LIN {X 0,Y 490.611,Z 701.735,A -85,B 0,C 180,E1 -6449.611,E2 -6449.611} C_VEL
LIN {X 0,Y 490.925,Z 689.002,A -85,B 0,C 180,E1 -6450.162,E2 -6450.162} C_VEL
LIN {X 0,Y 491.127,Z 676.229,A -85,B 0,C 180,E1 -6450.536,E2 -6450.536} C_VEL
LIN {X 0,Y 491.315,Z 653.215,A -85,B 0,C 180,E1 -6450.913,E2 -6450.913} C_VEL
LIN {X 0,Y 491.695,Z 579.169,A -85,B 0,C 180,E1 -6452.03,E2 -6452.03} C_VEL
LIN {X 0,Y 489.54,Z 572.056,A -85,B 0,C 180,E1 -6452.216,E2 -6452.216} C_VEL
LIN {X 0,Y 488.77,Z 569.605,A -85,B 0,C 180,E1 -6452.285,E2 -6452.285} C_VEL
LIN {X 0,Y 488.731,Z 569.605,A -85,B 0,C 180,E1 -6455.353,E2 -6455.353} C_VEL
LIN {X 0,Y 488.692,Z 569.612,A -85,B 0,C 180,E1 -6458.043,E2 -6458.043} C_VEL
LIN {X 0,Y 488.737,Z 569.609,A -85,B 0,C 180,E1 -6460.686,E2 -6460.686} C_VEL
LIN {X 0,Y 488.723,Z 569.605,A -85,B 0,C 180,E1 -6463.285,E2 -6463.285} C_VEL
LIN {X 0,Y 488.731,Z 569.605,A -85,B 0,C 180,E1 -6465.85,E2 -6465.85} C_VEL
LIN {X 0,Y 488.823,Z 569.598,A -85,B 0,C 180,E1 -6468.388,E2 -6468.388} C_VEL
LIN {X 0,Y 488.809,Z 569.594,A -85,B 0,C 180,E1 -6471.733,E2 -6471.733} C_VEL
LIN {X 0,Y 488.861,Z 569.591,A -85,B 0,C 180,E1 -6474.224,E2 -6474.224} C_VEL
LIN {X 0,Y 488.952,Z 569.573,A -85,B 0,C 180,E1 -6477.529,E2 -6477.529} C_VEL
LIN {X 0,Y 488.959,Z 569.576,A -85,B 0,C 180,E1 -6480,E2 -6480} C_VEL
LIN {X 0,Y 488.952,Z 569.583,A -85,B 0,C 180,E1 -6482.471,E2 -6482.471} C_VEL
LIN {X 0,Y 488.863,Z 569.586,A -85,B 0,C 180,E1 -6485.776,E2 -6485.776} C_VEL
LIN {X 0,Y 488.809,Z 569.595,A -85,B 0,C 180,E1 -6488.267,E2 -6488.267} C_VEL
LIN {X 0,Y 488.821,Z 569.589,A -85,B 0,C 180,E1 -6491.612,E2 -6491.612} C_VEL
LIN {X 0,Y 488.755,Z 569.599,A -85,B 0,C 180,E1 -6495.001,E2 -6495.001} C_VEL
LIN {X 0,Y 488.745,Z 569.604,A -85,B 0,C 180,E1 -6498.443,E2 -6498.443} C_VEL
LIN {X 0,Y 488.703,Z 569.606,A -85,B 0,C 180,E1 -6501.071,E2 -6501.071} C_VEL
LIN {X 0,Y 488.692,Z 569.605,A -85,B 0,C 180,E1 -6503.746,E2 -6503.746} C_VEL
LIN {X 0,Y 488.791,Z 569.595,A -85,B 0,C 180,E1 -6506.946,E2 -6506.946} C_VEL
LIN {X 0,Y 488.712,Z 569.61,A -85,B 0,C 180,E1 -6510.366,E2 -6510.366} C_VEL
LIN {X 0,Y 488.729,Z 569.601,A -85,B 0,C 180,E1 -6513.485,E2 -6513.485} C_VEL
LIN {X 0,Y 488.683,Z 569.614,A -85,B 0,C 180,E1 -6516.357,E2 -6516.357} C_VEL
LIN {X 0,Y 488.743,Z 569.6,A -85,B 0,C 180,E1 -6519.25,E2 -6519.25} C_VEL
LIN {X 0,Y 488.73,Z 569.61,A -85,B 0,C 180,E1 -6522.522,E2 -6522.522} C_VEL
LIN {X 0,Y 488.707,Z 569.607,A -85,B 0,C 180,E1 -6525.199,E2 -6525.199} C_VEL
LIN {X 0,Y 488.705,Z 569.613,A -85,B 0,C 180,E1 -6528.401,E2 -6528.401} C_VEL
LIN {X 0,Y 488.739,Z 569.605,A -85,B 0,C 180,E1 -6530.943,E2 -6530.943} C_VEL
LIN {X 0,Y 488.677,Z 569.611,A -85,B 0,C 180,E1 -6533.869,E2 -6533.869} C_VEL
LIN {X 0,Y 488.737,Z 569.606,A -85,B 0,C 180,E1 -6536.878,E2 -6536.878} C_VEL
LIN {X 0,Y 488.723,Z 569.607,A -85,B 0,C 180,E1 -6539.782,E2 -6539.782} C_VEL
LIN {X 0,Y 488.776,Z 569.651,A -85,B 0,C 180,E1 -6542.403,E2 -6542.403} C_VEL
LIN {X 0,Y 491.204,Z 581.744,A -85,B 0,C 180,E1 -6544.341,E2 -6544.341} C_VEL
LIN {X 0,Y 491.299,Z 586.393,A -85,B 0,C 180,E1 -6545.04,E2 -6545.04} C_VEL
LIN {X 0,Y 490.577,Z 606.107,A -85,B 0,C 180,E1 -6547.911,E2 -6547.911} C_VEL
LIN {X 0,Y 489.918,Z 627.979,A -85,B 0,C 180,E1 -6551.054,E2 -6551.054} C_VEL
LIN {X 0,Y 489.406,Z 646.726,A -85,B 0,C 180,E1 -6553.716,E2 -6553.716} C_VEL
LIN {X 0,Y 491.604,Z 665.305,A -85,B 0,C 180,E1 -6554.08,E2 -6554.08} C_VEL
LIN {X 0,Y 490.987,Z 757.207,A -85,B 0,C 180,E1 -6555.467,E2 -6555.467} C_VEL
LIN {X 0,Y 490.609,Z 771.003,A -85,B 0,C 180,E1 -6555.853,E2 -6555.853} C_VEL
LIN {X 0,Y 490.32,Z 783.46,A -85,B 0,C 180,E1 -6556.373,E2 -6556.373} C_VEL
LIN {X 0,Y 489.881,Z 795.901,A -85,B 0,C 180,E1 -6557.078,E2 -6557.078} C_VEL
LIN {X 0,Y 489.518,Z 806.944,A -85,B 0,C 180,E1 -6557.88,E2 -6557.88} C_VEL
LIN {X 0,Y 489.111,Z 817.345,A -85,B 0,C 180,E1 -6558.815,E2 -6558.815} C_VEL
LIN {X 0,Y 488.757,Z 826.697,A -85,B 0,C 180,E1 -6559.855,E2 -6559.855} C_VEL
LIN {X 0,Y 488.433,Z 835.805,A -85,B 0,C 180,E1 -6561.102,E2 -6561.102} C_VEL
LIN {X 0,Y 488.22,Z 843.153,A -85,B 0,C 180,E1 -6562.348,E2 -6562.348} C_VEL
LIN {X 0,Y 488.081,Z 848.576,A -85,B 0,C 180,E1 -6563.489,E2 -6563.489} C_VEL
LIN {X 0,Y 488.065,Z 852.942,A -85,B 0,C 180,E1 -6564.629,E2 -6564.629} C_VEL
LIN {X 0,Y 488.042,Z 856.64,A -85,B 0,C 180,E1 -6565.871,E2 -6565.871} C_VEL
LIN {X 0,Y 487.974,Z 858.545,A -85,B 0,C 180,E1 -6566.697,E2 -6566.697} C_VEL
LIN {X 0,Y 487.988,Z 859.977,A -85,B 0,C 180,E1 -6567.524,E2 -6567.524} C_VEL
LIN {X 0,Y 487.853,Z 861.615,A -85,B 0,C 180,E1 -6569.175,E2 -6569.175} C_VEL
LIN {X 0,Y 487.847,Z 861.844,A -85,B 0,C 180,E1 -6570,E2 -6570} C_VEL
LIN {X 0,Y 487.852,Z 861.63,A -85,B 0,C 180,E1 -6570.825,E2 -6570.825} C_VEL
LIN {X 0,Y 487.988,Z 860.021,A -85,B 0,C 180,E1 -6572.476,E2 -6572.476} C_VEL
LIN {X 0,Y 487.973,Z 858.603,A -85,B 0,C 180,E1 -6573.303,E2 -6573.303} C_VEL
LIN {X 0,Y 487.959,Z 855.624,A -85,B 0,C 180,E1 -6574.543,E2 -6574.543} C_VEL
LIN {X 0,Y 488.08,Z 851.599,A -85,B 0,C 180,E1 -6575.785,E2 -6575.785} C_VEL
LIN {X 0,Y 488.181,Z 845.387,A -85,B 0,C 180,E1 -6577.236,E2 -6577.236} C_VEL
LIN {X 0,Y 488.379,Z 838.614,A -85,B 0,C 180,E1 -6578.482,E2 -6578.482} C_VEL
LIN {X 0,Y 488.615,Z 830.213,A -85,B 0,C 180,E1 -6579.73,E2 -6579.73} C_VEL
LIN {X 0,Y 488.939,Z 821.594,A -85,B 0,C 180,E1 -6580.769,E2 -6580.769} C_VEL
LIN {X 0,Y 489.324,Z 810.96,A -85,B 0,C 180,E1 -6581.81,E2 -6581.81} C_VEL
LIN {X 0,Y 489.743,Z 799.505,A -85,B 0,C 180,E1 -6582.709,E2 -6582.709} C_VEL
LIN {X 0,Y 490.111,Z 788.898,A -85,B 0,C 180,E1 -6583.369,E2 -6583.369} C_VEL
LIN {X 0,Y 490.533,Z 776.972,A -85,B 0,C 180,E1 -6583.938,E2 -6583.938} C_VEL
LIN {X 0,Y 490.91,Z 764.13,A -85,B 0,C 180,E1 -6584.376,E2 -6584.376} C_VEL
LIN {X 0,Y 491.134,Z 750.796,A -85,B 0,C 180,E1 -6584.661,E2 -6584.661} C_VEL
LIN {X 0,Y 491.593,Z 661.443,A -85,B 0,C 180,E1 -6585.99,E2 -6585.99} C_VEL
LIN {X 0,Y 489.745,Z 646.4,A -85,B 0,C 180,E1 -6586.299,E2 -6586.299} C_VEL
LIN {X 0,Y 490.543,Z 619.4,A -85,B 0,C 180,E1 -6589.674,E2 -6589.674} C_VEL
LIN {X 0,Y 491.408,Z 595.344,A -85,B 0,C 180,E1 -6592.714,E2 -6592.714} C_VEL
LIN {X 0,Y 491.831,Z 584.522,A -85,B 0,C 180,E1 -6594.096,E2 -6594.096} C_VEL
LIN {X 0,Y 489.098,Z 571.021,A -85,B 0,C 180,E1 -6595.992,E2 -6595.992} C_VEL
LIN {X 0,Y 488.783,Z 569.602,A -85,B 0,C 180,E1 -6596.24,E2 -6596.24} C_VEL
LIN {X 0,Y 488.723,Z 569.607,A -85,B 0,C 180,E1 -6599.27,E2 -6599.27} C_VEL
LIN {X 0,Y 488.703,Z 569.613,A -85,B 0,C 180,E1 -6602.146,E2 -6602.146} C_VEL
LIN {X 0,Y 488.722,Z 569.604,A -85,B 0,C 180,E1 -6605.114,E2 -6605.114} C_VEL
LIN {X 0,Y 488.68,Z 569.612,A -85,B 0,C 180,E1 -6608.199,E2 -6608.199} C_VEL
LIN {X 0,Y 488.746,Z 569.604,A -85,B 0,C 180,E1 -6610.348,E2 -6610.348} C_VEL
LIN {X 0,Y 488.683,Z 569.61,A -85,B 0,C 180,E1 -6613.653,E2 -6613.653} C_VEL
LIN {X 0,Y 488.712,Z 569.61,A -85,B 0,C 180,E1 -6616.348,E2 -6616.348} C_VEL
LIN {X 0,Y 488.731,Z 569.603,A -85,B 0,C 180,E1 -6619.676,E2 -6619.676} C_VEL
LIN {X 0,Y 488.678,Z 569.617,A -85,B 0,C 180,E1 -6622.276,E2 -6622.276} C_VEL
LIN {X 0,Y 488.722,Z 569.597,A -85,B 0,C 180,E1 -6625.051,E2 -6625.051} C_VEL
LIN {X 0,Y 488.699,Z 569.61,A -85,B 0,C 180,E1 -6628.045,E2 -6628.045} C_VEL
LIN {X 0,Y 488.726,Z 569.599,A -85,B 0,C 180,E1 -6630.73,E2 -6630.73} C_VEL
LIN {X 0,Y 488.758,Z 569.598,A -85,B 0,C 180,E1 -6633.528,E2 -6633.528} C_VEL
LIN {X 0,Y 488.685,Z 569.611,A -85,B 0,C 180,E1 -6636.254,E2 -6636.254} C_VEL
LIN {X 0,Y 488.737,Z 569.601,A -85,B 0,C 180,E1 -6639.175,E2 -6639.175} C_VEL
LIN {X 0,Y 488.75,Z 569.599,A -85,B 0,C 180,E1 -6641.627,E2 -6641.627} C_VEL
LIN {X 0,Y 488.752,Z 569.599,A -85,B 0,C 180,E1 -6644.999,E2 -6644.999} C_VEL
LIN {X 0,Y 488.798,Z 569.6,A -85,B 0,C 180,E1 -6648.387,E2 -6648.387} C_VEL
LIN {X 0,Y 488.808,Z 569.585,A -85,B 0,C 180,E1 -6651.733,E2 -6651.733} C_VEL
LIN {X 0,Y 488.864,Z 569.587,A -85,B 0,C 180,E1 -6654.224,E2 -6654.224} C_VEL
LIN {X 0,Y 488.952,Z 569.568,A -85,B 0,C 180,E1 -6657.529,E2 -6657.529} C_VEL
LIN {X 0,Y 488.959,Z 569.57,A -85,B 0,C 180,E1 -6660,E2 -6660} C_VEL
LIN {X 0,Y 488.952,Z 569.579,A -85,B 0,C 180,E1 -6662.471,E2 -6662.471} C_VEL
LIN {X 0,Y 488.855,Z 569.577,A -85,B 0,C 180,E1 -6665.776,E2 -6665.776} C_VEL
LIN {X 0,Y 488.808,Z 569.593,A -85,B 0,C 180,E1 -6668.267,E2 -6668.267} C_VEL
LIN {X 0,Y 488.798,Z 569.588,A -85,B 0,C 180,E1 -6671.613,E2 -6671.613} C_VEL
LIN {X 0,Y 488.752,Z 569.607,A -85,B 0,C 180,E1 -6675.001,E2 -6675.001} C_VEL
LIN {X 0,Y 488.745,Z 569.599,A -85,B 0,C 180,E1 -6678.443,E2 -6678.443} C_VEL
LIN {X 0,Y 488.697,Z 569.614,A -85,B 0,C 180,E1 -6681.071,E2 -6681.071} C_VEL
LIN {X 0,Y 488.684,Z 569.605,A -85,B 0,C 180,E1 -6683.746,E2 -6683.746} C_VEL
LIN {X 0,Y 488.791,Z 569.6,A -85,B 0,C 180,E1 -6686.946,E2 -6686.946} C_VEL
LIN {X 0,Y 488.711,Z 569.601,A -85,B 0,C 180,E1 -6690.365,E2 -6690.365} C_VEL
LIN {X 0,Y 488.729,Z 569.603,A -85,B 0,C 180,E1 -6693.485,E2 -6693.485} C_VEL
LIN {X 0,Y 488.683,Z 569.608,A -85,B 0,C 180,E1 -6696.357,E2 -6696.357} C_VEL
LIN {X 0,Y 488.724,Z 569.61,A -85,B 0,C 180,E1 -6699.252,E2 -6699.252} C_VEL
LIN {X 0,Y 488.69,Z 569.596,A -85,B 0,C 180,E1 -6702.526,E2 -6702.526} C_VEL
LIN {X 0,Y 488.707,Z 569.612,A -85,B 0,C 180,E1 -6705.199,E2 -6705.199} C_VEL
LIN {X 0,Y 488.704,Z 569.602,A -85,B 0,C 180,E1 -6708.585,E2 -6708.585} C_VEL
LIN {X 0,Y 488.702,Z 569.61,A -85,B 0,C 180,E1 -6710.948,E2 -6710.948} C_VEL
LIN {X 0,Y 488.683,Z 569.611,A -85,B 0,C 180,E1 -6713.869,E2 -6713.869} C_VEL
LIN {X 0,Y 488.737,Z 569.604,A -85,B 0,C 180,E1 -6716.878,E2 -6716.878} C_VEL
LIN {X 0,Y 488.723,Z 569.61,A -85,B 0,C 180,E1 -6719.781,E2 -6719.781} C_VEL
LIN {X 0,Y 488.755,Z 569.621,A -85,B 0,C 180,E1 -6721.82,E2 -6721.82} C_VEL
LIN {X 0,Y 491.447,Z 578.092,A -85,B 0,C 180,E1 -6722.042,E2 -6722.042} C_VEL
LIN {X 0,Y 491.827,Z 581.103,A -85,B 0,C 180,E1 -6722.101,E2 -6722.101} C_VEL
LIN {X 0,Y 491.734,Z 596.411,A -85,B 0,C 180,E1 -6722.326,E2 -6722.326} C_VEL
LIN {X 0,Y 491.108,Z 602.256,A -85,B 0,C 180,E1 -6722.392,E2 -6722.392} C_VEL
LIN {X 0,Y 485.37,Z 621.251,A -85,B 0,C 180,E1 -6722.482,E2 -6722.482} C_VEL
LIN {X 0,Y 484.685,Z 627.099,A -85,B 0,C 180,E1 -6722.547,E2 -6722.547} C_VEL
LIN {X 0,Y 484.361,Z 674.303,A -85,B 0,C 180,E1 -6723.27,E2 -6723.27} C_VEL
LIN {X 0,Y 484.136,Z 686.741,A -85,B 0,C 180,E1 -6723.605,E2 -6723.605} C_VEL
LIN {X 0,Y 483.895,Z 699.222,A -85,B 0,C 180,E1 -6724.112,E2 -6724.112} C_VEL
LIN {X 0,Y 483.572,Z 710.665,A -85,B 0,C 180,E1 -6724.745,E2 -6724.745} C_VEL
LIN {X 0,Y 483.138,Z 721.486,A -85,B 0,C 180,E1 -6725.508,E2 -6725.508} C_VEL
LIN {X 0,Y 482.69,Z 731.974,A -85,B 0,C 180,E1 -6726.433,E2 -6726.433} C_VEL
LIN {X 0,Y 482.283,Z 741.728,A -85,B 0,C 180,E1 -6727.51,E2 -6727.51} C_VEL
LIN {X 0,Y 481.943,Z 749.915,A -85,B 0,C 180,E1 -6728.62,E2 -6728.62} C_VEL
LIN {X 0,Y 481.552,Z 757.827,A -85,B 0,C 180,E1 -6729.943,E2 -6729.943} C_VEL
LIN {X 0,Y 481.346,Z 764.048,A -85,B 0,C 180,E1 -6731.264,E2 -6731.264} C_VEL
LIN {X 0,Y 481.157,Z 768.904,A -85,B 0,C 180,E1 -6732.577,E2 -6732.577} C_VEL
LIN {X 0,Y 481.036,Z 772.562,A -85,B 0,C 180,E1 -6733.884,E2 -6733.884} C_VEL
LIN {X 0,Y 480.962,Z 774.42,A -85,B 0,C 180,E1 -6734.751,E2 -6734.751} C_VEL
LIN {X 0,Y 480.908,Z 775.786,A -85,B 0,C 180,E1 -6735.615,E2 -6735.615} C_VEL
LIN {X 0,Y 480.869,Z 777.298,A -85,B 0,C 180,E1 -6737.337,E2 -6737.337} C_VEL
LIN {X 0,Y 480.912,Z 777.394,A -85,B 0,C 180,E1 -6738.275,E2 -6738.275} C_VEL
LIN {X 0,Y 480.876,Z 776.456,A -85,B 0,C 180,E1 -6739.899,E2 -6739.899} C_VEL
LIN {X 0,Y 480.912,Z 775.377,A -85,B 0,C 180,E1 -6740.75,E2 -6740.75} C_VEL
LIN {X 0,Y 480.968,Z 773.857,A -85,B 0,C 180,E1 -6741.598,E2 -6741.598} C_VEL
LIN {X 0,Y 481.149,Z 770.786,A -85,B 0,C 180,E1 -6742.868,E2 -6742.868} C_VEL
LIN {X 0,Y 481.199,Z 766.705,A -85,B 0,C 180,E1 -6744.132,E2 -6744.132} C_VEL
LIN {X 0,Y 481.409,Z 760.498,A -85,B 0,C 180,E1 -6745.604,E2 -6745.604} C_VEL
LIN {X 0,Y 481.708,Z 753.684,A -85,B 0,C 180,E1 -6746.864,E2 -6746.864} C_VEL
LIN {X 0,Y 482.052,Z 745.219,A -85,B 0,C 180,E1 -6748.12,E2 -6748.12} C_VEL
LIN {X 0,Y 482.485,Z 736.553,A -85,B 0,C 180,E1 -6749.165,E2 -6749.165} C_VEL
LIN {X 0,Y 482.813,Z 727.09,A -85,B 0,C 180,E1 -6750.104,E2 -6750.104} C_VEL
LIN {X 0,Y 483.274,Z 716.632,A -85,B 0,C 180,E1 -6750.937,E2 -6750.937} C_VEL
LIN {X 0,Y 483.739,Z 705.073,A -85,B 0,C 180,E1 -6751.665,E2 -6751.665} C_VEL
LIN {X 0,Y 483.994,Z 693.264,A -85,B 0,C 180,E1 -6752.236,E2 -6752.236} C_VEL
LIN {X 0,Y 484.251,Z 680.14,A -85,B 0,C 180,E1 -6752.677,E2 -6752.677} C_VEL
LIN {X 0,Y 484.424,Z 665.875,A -85,B 0,C 180,E1 -6752.963,E2 -6752.963} C_VEL
LIN {X 0,Y 484.994,Z 579.93,A -85,B 0,C 180,E1 -6754.242,E2 -6754.242} C_VEL
LIN {X 0,Y 481.732,Z 570.675,A -85,B 0,C 180,E1 -6754.498,E2 -6754.498} C_VEL
LIN {X 0,Y 481.779,Z 570.471,A -85,B 0,C 180,E1 -6756.702,E2 -6756.702} C_VEL
LIN {X 0,Y 481.735,Z 570.475,A -85,B 0,C 180,E1 -6759.234,E2 -6759.234} C_VEL
LIN {X 0,Y 481.777,Z 570.474,A -85,B 0,C 180,E1 -6762.211,E2 -6762.211} C_VEL
LIN {X 0,Y 481.728,Z 570.478,A -85,B 0,C 180,E1 -6765.658,E2 -6765.658} C_VEL
LIN {X 0,Y 481.714,Z 570.477,A -85,B 0,C 180,E1 -6768.721,E2 -6768.721} C_VEL
LIN {X 0,Y 481.646,Z 570.485,A -85,B 0,C 180,E1 -6771.394,E2 -6771.394} C_VEL
LIN {X 0,Y 481.658,Z 570.491,A -85,B 0,C 180,E1 -6774.113,E2 -6774.113} C_VEL
LIN {X 0,Y 481.747,Z 570.474,A -85,B 0,C 180,E1 -6777.139,E2 -6777.139} C_VEL
LIN {X 0,Y 481.698,Z 570.484,A -85,B 0,C 180,E1 -6779.581,E2 -6779.581} C_VEL
LIN {X 0,Y 484.986,Z 579.827,A -85,B 0,C 180,E1 -6779.846,E2 -6779.846} C_VEL
LIN {X 0,Y 484.24,Z 674.779,A -85,B 0,C 180,E1 -6781.308,E2 -6781.308} C_VEL
LIN {X 0,Y 484.063,Z 688.668,A -85,B 0,C 180,E1 -6781.709,E2 -6781.709} C_VEL
LIN {X 0,Y 483.747,Z 701.601,A -85,B 0,C 180,E1 -6782.269,E2 -6782.269} C_VEL
LIN {X 0,Y 483.34,Z 713.832,A -85,B 0,C 180,E1 -6782.992,E2 -6782.992} C_VEL
LIN {X 0,Y 482.933,Z 725.238,A -85,B 0,C 180,E1 -6783.859,E2 -6783.859} C_VEL
LIN {X 0,Y 482.522,Z 735.559,A -85,B 0,C 180,E1 -6784.849,E2 -6784.849} C_VEL
LIN {X 0,Y 482.095,Z 744.579,A -85,B 0,C 180,E1 -6785.914,E2 -6785.914} C_VEL
LIN {X 0,Y 481.803,Z 752.062,A -85,B 0,C 180,E1 -6786.991,E2 -6786.991} C_VEL
LIN {X 0,Y 481.518,Z 758.715,A -85,B 0,C 180,E1 -6788.154,E2 -6788.154} C_VEL
LIN {X 0,Y 481.362,Z 764.062,A -85,B 0,C 180,E1 -6789.302,E2 -6789.302} C_VEL
LIN {X 0,Y 481.147,Z 768.812,A -85,B 0,C 180,E1 -6790.575,E2 -6790.575} C_VEL
LIN {X 0,Y 480.991,Z 773.335,A -85,B 0,C 180,E1 -6792.23,E2 -6792.23} C_VEL
LIN {X 0,Y 480.89,Z 775.492,A -85,B 0,C 180,E1 -6793.383,E2 -6793.383} C_VEL
LIN {X 0,Y 480.844,Z 776.858,A -85,B 0,C 180,E1 -6794.551,E2 -6794.551} C_VEL
LIN {X 0,Y 480.797,Z 777.469,A -85,B 0,C 180,E1 -6795.744,E2 -6795.744} C_VEL
LIN {X 0,Y 480.843,Z 777.285,A -85,B 0,C 180,E1 -6796.952,E2 -6796.952} C_VEL
LIN {X 0,Y 480.888,Z 776.261,A -85,B 0,C 180,E1 -6798.187,E2 -6798.187} C_VEL
LIN {X 0,Y 480.936,Z 774.305,A -85,B 0,C 180,E1 -6799.452,E2 -6799.452} C_VEL
LIN {X 0,Y 481.107,Z 770.315,A -85,B 0,C 180,E1 -6801.087,E2 -6801.087} C_VEL
LIN {X 0,Y 481.297,Z 765.708,A -85,B 0,C 180,E1 -6802.436,E2 -6802.436} C_VEL
LIN {X 0,Y 481.517,Z 759.399,A -85,B 0,C 180,E1 -6803.852,E2 -6803.852} C_VEL
LIN {X 0,Y 481.769,Z 752.609,A -85,B 0,C 180,E1 -6805.058,E2 -6805.058} C_VEL
LIN {X 0,Y 482.179,Z 744.851,A -85,B 0,C 180,E1 -6806.179,E2 -6806.179} C_VEL
LIN {X 0,Y 482.503,Z 735.703,A -85,B 0,C 180,E1 -6807.265,E2 -6807.265} C_VEL
LIN {X 0,Y 482.929,Z 726.436,A -85,B 0,C 180,E1 -6808.16,E2 -6808.16} C_VEL
LIN {X 0,Y 483.333,Z 715.731,A -85,B 0,C 180,E1 -6808.998,E2 -6808.998} C_VEL
LIN {X 0,Y 483.686,Z 703.676,A -85,B 0,C 180,E1 -6809.734,E2 -6809.734} C_VEL
LIN {X 0,Y 484.048,Z 691.314,A -85,B 0,C 180,E1 -6810.299,E2 -6810.299} C_VEL
LIN {X 0,Y 484.268,Z 678.506,A -85,B 0,C 180,E1 -6810.702,E2 -6810.702} C_VEL
LIN {X 0,Y 484.402,Z 661.544,A -85,B 0,C 180,E1 -6811.009,E2 -6811.009} C_VEL
LIN {X 0,Y 484.939,Z 580.221,A -85,B 0,C 180,E1 -6812.254,E2 -6812.254} C_VEL
LIN {X 0,Y 481.746,Z 570.48,A -85,B 0,C 180,E1 -6812.533,E2 -6812.533} C_VEL
LIN {X 0,Y 481.669,Z 570.486,A -85,B 0,C 180,E1 -6815.886,E2 -6815.886} C_VEL
LIN {X 0,Y 481.693,Z 570.483,A -85,B 0,C 180,E1 -6819.027,E2 -6819.027} C_VEL
LIN {X 0,Y 481.698,Z 570.483,A -85,B 0,C 180,E1 -6822.158,E2 -6822.158} C_VEL
LIN {X 0,Y 481.733,Z 570.481,A -85,B 0,C 180,E1 -6824.775,E2 -6824.775} C_VEL
LIN {X 0,Y 481.786,Z 570.473,A -85,B 0,C 180,E1 -6828.216,E2 -6828.216} C_VEL
LIN {X 0,Y 481.754,Z 570.472,A -85,B 0,C 180,E1 -6831.612,E2 -6831.612} C_VEL
LIN {X 0,Y 481.819,Z 570.467,A -85,B 0,C 180,E1 -6834.14,E2 -6834.14} C_VEL
LIN {X 0,Y 481.919,Z 570.449,A -85,B 0,C 180,E1 -6837.493,E2 -6837.493} C_VEL
LIN {X 0,Y 481.93,Z 570.452,A -85,B 0,C 180,E1 -6840,E2 -6840} C_VEL
LIN {X 0,Y 481.919,Z 570.458,A -85,B 0,C 180,E1 -6842.508,E2 -6842.508} C_VEL
LIN {X 0,Y 481.821,Z 570.464,A -85,B 0,C 180,E1 -6845.86,E2 -6845.86} C_VEL
LIN {X 0,Y 481.754,Z 570.476,A -85,B 0,C 180,E1 -6848.388,E2 -6848.388} C_VEL
LIN {X 0,Y 481.786,Z 570.466,A -85,B 0,C 180,E1 -6851.784,E2 -6851.784} C_VEL
LIN {X 0,Y 481.734,Z 570.472,A -85,B 0,C 180,E1 -6855.225,E2 -6855.225} C_VEL
LIN {X 0,Y 481.703,Z 570.481,A -85,B 0,C 180,E1 -6858.722,E2 -6858.722} C_VEL
LIN {X 0,Y 481.645,Z 570.483,A -85,B 0,C 180,E1 -6861.395,E2 -6861.395} C_VEL
LIN {X 0,Y 481.674,Z 570.482,A -85,B 0,C 180,E1 -6864.113,E2 -6864.113} C_VEL
LIN {X 0,Y 481.744,Z 570.471,A -85,B 0,C 180,E1 -6867.141,E2 -6867.141} C_VEL
LIN {X 0,Y 481.681,Z 570.481,A -85,B 0,C 180,E1 -6869.741,E2 -6869.741} C_VEL
LIN {X 0,Y 481.666,Z 570.487,A -85,B 0,C 180,E1 -6872.675,E2 -6872.675} C_VEL
LIN {X 0,Y 481.637,Z 570.487,A -85,B 0,C 180,E1 -6875.71,E2 -6875.71} C_VEL
LIN {X 0,Y 481.714,Z 570.476,A -85,B 0,C 180,E1 -6879.355,E2 -6879.355} C_VEL
LIN {X 0,Y 481.67,Z 570.485,A -85,B 0,C 180,E1 -6882.159,E2 -6882.159} C_VEL
LIN {X 0,Y 481.656,Z 570.491,A -85,B 0,C 180,E1 -6884.458,E2 -6884.458} C_VEL
LIN {X 0,Y 481.644,Z 570.488,A -85,B 0,C 180,E1 -6887.84,E2 -6887.84} C_VEL
LIN {X 0,Y 481.712,Z 570.483,A -85,B 0,C 180,E1 -6890.647,E2 -6890.647} C_VEL
LIN {X 0,Y 481.636,Z 570.493,A -85,B 0,C 180,E1 -6894.291,E2 -6894.291} C_VEL
LIN {X 0,Y 481.671,Z 570.485,A -85,B 0,C 180,E1 -6897.327,E2 -6897.327} C_VEL
LIN {X 0,Y 481.678,Z 570.487,A -85,B 0,C 180,E1 -6900.26,E2 -6900.26} C_VEL
LIN {X 0,Y 481.731,Z 570.549,A -85,B 0,C 180,E1 -6902.193,E2 -6902.193} C_VEL
LIN {X 0,Y 484.184,Z 582.746,A -85,B 0,C 180,E1 -6904.187,E2 -6904.187} C_VEL
LIN {X 0,Y 484.403,Z 587.321,A -85,B 0,C 180,E1 -6904.89,E2 -6904.89} C_VEL
LIN {X 0,Y 483.618,Z 606.955,A -85,B 0,C 180,E1 -6907.801,E2 -6907.801} C_VEL
LIN {X 0,Y 482.904,Z 627.763,A -85,B 0,C 180,E1 -6910.834,E2 -6910.834} C_VEL
LIN {X 0,Y 482.374,Z 646.048,A -85,B 0,C 180,E1 -6913.474,E2 -6913.474} C_VEL
LIN {X 0,Y 484.761,Z 665.54,A -85,B 0,C 180,E1 -6913.862,E2 -6913.862} C_VEL
LIN {X 0,Y 484.094,Z 756.265,A -85,B 0,C 180,E1 -6915.255,E2 -6915.255} C_VEL
LIN {X 0,Y 483.728,Z 770.154,A -85,B 0,C 180,E1 -6915.647,E2 -6915.647} C_VEL
LIN {X 0,Y 483.361,Z 782.664,A -85,B 0,C 180,E1 -6916.173,E2 -6916.173} C_VEL
LIN {X 0,Y 482.907,Z 795.142,A -85,B 0,C 180,E1 -6916.888,E2 -6916.888} C_VEL
LIN {X 0,Y 482.554,Z 805.647,A -85,B 0,C 180,E1 -6917.656,E2 -6917.656} C_VEL
LIN {X 0,Y 482.073,Z 815.544,A -85,B 0,C 180,E1 -6918.543,E2 -6918.543} C_VEL
LIN {X 0,Y 481.752,Z 824.27,A -85,B 0,C 180,E1 -6919.493,E2 -6919.493} C_VEL
LIN {X 0,Y 481.469,Z 832.323,A -85,B 0,C 180,E1 -6920.549,E2 -6920.549} C_VEL
LIN {X 0,Y 481.243,Z 840.204,A -85,B 0,C 180,E1 -6921.814,E2 -6921.814} C_VEL
LIN {X 0,Y 481.048,Z 847.457,A -85,B 0,C 180,E1 -6923.288,E2 -6923.288} C_VEL
LIN {X 0,Y 481.002,Z 852.299,A -85,B 0,C 180,E1 -6924.55,E2 -6924.55} C_VEL
LIN {X 0,Y 480.938,Z 856.002,A -85,B 0,C 180,E1 -6925.81,E2 -6925.81} C_VEL
LIN {X 0,Y 480.904,Z 857.915,A -85,B 0,C 180,E1 -6926.649,E2 -6926.649} C_VEL
LIN {X 0,Y 480.925,Z 859.352,A -85,B 0,C 180,E1 -6927.487,E2 -6927.487} C_VEL
LIN {X 0,Y 480.78,Z 860.998,A -85,B 0,C 180,E1 -6929.162,E2 -6929.162} C_VEL
LIN {X 0,Y 480.774,Z 861.229,A -85,B 0,C 180,E1 -6930,E2 -6930} C_VEL
LIN {X 0,Y 480.826,Z 860.409,A -85,B 0,C 180,E1 -6931.675,E2 -6931.675} C_VEL
LIN {X 0,Y 480.925,Z 859.411,A -85,B 0,C 180,E1 -6932.513,E2 -6932.513} C_VEL
LIN {X 0,Y 480.902,Z 857.992,A -85,B 0,C 180,E1 -6933.351,E2 -6933.351} C_VEL
LIN {X 0,Y 480.871,Z 855.01,A -85,B 0,C 180,E1 -6934.61,E2 -6934.61} C_VEL
LIN {X 0,Y 480.977,Z 850.981,A -85,B 0,C 180,E1 -6935.871,E2 -6935.871} C_VEL
LIN {X 0,Y 481.107,Z 844.765,A -85,B 0,C 180,E1 -6937.343,E2 -6937.343} C_VEL
LIN {X 0,Y 481.313,Z 837.985,A -85,B 0,C 180,E1 -6938.607,E2 -6938.607} C_VEL
LIN {X 0,Y 481.552,Z 829.576,A -85,B 0,C 180,E1 -6939.874,E2 -6939.874} C_VEL
LIN {X 0,Y 481.906,Z 820.946,A -85,B 0,C 180,E1 -6940.928,E2 -6940.928} C_VEL
LIN {X 0,Y 482.329,Z 810.481,A -85,B 0,C 180,E1 -6941.968,E2 -6941.968} C_VEL
LIN {X 0,Y 482.723,Z 800.059,A -85,B 0,C 180,E1 -6942.806,E2 -6942.806} C_VEL
LIN {X 0,Y 483.165,Z 788.205,A -85,B 0,C 180,E1 -6943.565,E2 -6943.565} C_VEL
LIN {X 0,Y 483.613,Z 776.243,A -85,B 0,C 180,E1 -6944.142,E2 -6944.142} C_VEL
LIN {X 0,Y 483.999,Z 763.351,A -85,B 0,C 180,E1 -6944.586,E2 -6944.586} C_VEL
LIN {X 0,Y 484.251,Z 749.856,A -85,B 0,C 180,E1 -6944.874,E2 -6944.874} C_VEL
LIN {X 0,Y 484.699,Z 661.918,A -85,B 0,C 180,E1 -6946.207,E2 -6946.207} C_VEL
LIN {X 0,Y 482.739,Z 645.869,A -85,B 0,C 180,E1 -6946.536,E2 -6946.536} C_VEL
LIN {X 0,Y 483.569,Z 620.534,A -85,B 0,C 180,E1 -6949.749,E2 -6949.749} C_VEL
LIN {X 0,Y 484.554,Z 594.8,A -85,B 0,C 180,E1 -6953.054,E2 -6953.054} C_VEL
LIN {X 0,Y 484.924,Z 586.214,A -85,B 0,C 180,E1 -6954.168,E2 -6954.168} C_VEL
LIN {X 0,Y 483.32,Z 577.515,A -85,B 0,C 180,E1 -6955.396,E2 -6955.396} C_VEL
LIN {X 0,Y 481.737,Z 570.48,A -85,B 0,C 180,E1 -6956.42,E2 -6956.42} C_VEL
LIN {X 0,Y 481.678,Z 570.487,A -85,B 0,C 180,E1 -6959.74,E2 -6959.74} C_VEL
LIN {X 0,Y 481.671,Z 570.483,A -85,B 0,C 180,E1 -6962.673,E2 -6962.673} C_VEL
LIN {X 0,Y 481.642,Z 570.49,A -85,B 0,C 180,E1 -6965.708,E2 -6965.708} C_VEL
LIN {X 0,Y 481.711,Z 570.476,A -85,B 0,C 180,E1 -6969.353,E2 -6969.353} C_VEL
LIN {X 0,Y 481.645,Z 570.489,A -85,B 0,C 180,E1 -6972.16,E2 -6972.16} C_VEL
LIN {X 0,Y 481.656,Z 570.483,A -85,B 0,C 180,E1 -6975.542,E2 -6975.542} C_VEL
LIN {X 0,Y 481.668,Z 570.489,A -85,B 0,C 180,E1 -6978.084,E2 -6978.084} C_VEL
LIN {X 0,Y 481.698,Z 570.476,A -85,B 0,C 180,E1 -6981.143,E2 -6981.143} C_VEL
LIN {X 0,Y 481.662,Z 570.478,A -85,B 0,C 180,E1 -6984.794,E2 -6984.794} C_VEL
LIN {X 0,Y 481.666,Z 570.481,A -85,B 0,C 180,E1 -6987.325,E2 -6987.325} C_VEL
LIN {X 0,Y 481.681,Z 570.482,A -85,B 0,C 180,E1 -6990.259,E2 -6990.259} C_VEL
LIN {X 0,Y 481.744,Z 570.472,A -85,B 0,C 180,E1 -6993.112,E2 -6993.112} C_VEL
LIN {X 0,Y 481.668,Z 570.483,A -85,B 0,C 180,E1 -6995.886,E2 -6995.886} C_VEL
LIN {X 0,Y 481.693,Z 570.479,A -85,B 0,C 180,E1 -6999.027,E2 -6999.027} C_VEL
LIN {X 0,Y 481.698,Z 570.482,A -85,B 0,C 180,E1 -7002.158,E2 -7002.158} C_VEL
LIN {X 0,Y 481.732,Z 570.475,A -85,B 0,C 180,E1 -7004.775,E2 -7004.775} C_VEL
LIN {X 0,Y 481.742,Z 570.476,A -85,B 0,C 180,E1 -7008.215,E2 -7008.215} C_VEL
LIN {X 0,Y 481.754,Z 570.463,A -85,B 0,C 180,E1 -7011.612,E2 -7011.612} C_VEL
LIN {X 0,Y 481.822,Z 570.464,A -85,B 0,C 180,E1 -7014.14,E2 -7014.14} C_VEL
LIN {X 0,Y 481.919,Z 570.444,A -85,B 0,C 180,E1 -7017.492,E2 -7017.492} C_VEL
LIN {X 0,Y 481.93,Z 570.445,A -85,B 0,C 180,E1 -7020,E2 -7020} C_VEL
LIN {X 0,Y 481.919,Z 570.456,A -85,B 0,C 180,E1 -7022.508,E2 -7022.508} C_VEL
LIN {X 0,Y 481.814,Z 570.454,A -85,B 0,C 180,E1 -7025.86,E2 -7025.86} C_VEL
LIN {X 0,Y 481.754,Z 570.473,A -85,B 0,C 180,E1 -7028.388,E2 -7028.388} C_VEL
LIN {X 0,Y 481.743,Z 570.466,A -85,B 0,C 180,E1 -7031.785,E2 -7031.785} C_VEL
LIN {X 0,Y 481.732,Z 570.478,A -85,B 0,C 180,E1 -7035.225,E2 -7035.225} C_VEL
LIN {X 0,Y 481.703,Z 570.478,A -85,B 0,C 180,E1 -7038.722,E2 -7038.722} C_VEL
LIN {X 0,Y 481.636,Z 570.489,A -85,B 0,C 180,E1 -7041.395,E2 -7041.395} C_VEL
LIN {X 0,Y 481.668,Z 570.478,A -85,B 0,C 180,E1 -7044.114,E2 -7044.114} C_VEL
LIN {X 0,Y 481.744,Z 570.48,A -85,B 0,C 180,E1 -7047.141,E2 -7047.141} C_VEL
LIN {X 0,Y 481.681,Z 570.477,A -85,B 0,C 180,E1 -7049.741,E2 -7049.741} C_VEL
LIN {X 0,Y 481.666,Z 570.485,A -85,B 0,C 180,E1 -7052.675,E2 -7052.675} C_VEL
LIN {X 0,Y 481.636,Z 570.488,A -85,B 0,C 180,E1 -7055.71,E2 -7055.71} C_VEL
LIN {X 0,Y 481.666,Z 570.486,A -85,B 0,C 180,E1 -7058.86,E2 -7058.86} C_VEL
LIN {X 0,Y 481.657,Z 570.472,A -85,B 0,C 180,E1 -7061.915,E2 -7061.915} C_VEL
LIN {X 0,Y 481.655,Z 570.483,A -85,B 0,C 180,E1 -7064.458,E2 -7064.458} C_VEL
LIN {X 0,Y 481.643,Z 570.482,A -85,B 0,C 180,E1 -7067.84,E2 -7067.84} C_VEL
LIN {X 0,Y 481.677,Z 570.482,A -85,B 0,C 180,E1 -7070.652,E2 -7070.652} C_VEL
LIN {X 0,Y 481.629,Z 570.492,A -85,B 0,C 180,E1 -7073.376,E2 -7073.376} C_VEL
LIN {X 0,Y 481.708,Z 570.478,A -85,B 0,C 180,E1 -7076.331,E2 -7076.331} C_VEL
LIN {X 0,Y 481.65,Z 570.491,A -85,B 0,C 180,E1 -7079.418,E2 -7079.418} C_VEL
LIN {X 0,Y 481.732,Z 570.648,A -85,B 0,C 180,E1 -7081.58,E2 -7081.58} C_VEL
LIN {X 0,Y 484.862,Z 580.098,A -85,B 0,C 180,E1 -7081.84,E2 -7081.84} C_VEL
LIN {X 0,Y 484.739,Z 622.266,A -85,B 0,C 180,E1 -7082.475,E2 -7082.475} C_VEL
LIN {X 0,Y 484.685,Z 627.099,A -85,B 0,C 180,E1 -7082.547,E2 -7082.547} C_VEL
LIN {X 0,Y 484.027,Z 632.941,A -85,B 0,C 180,E1 -7082.612,E2 -7082.612} C_VEL
LIN {X 0,Y 478.374,Z 651.942,A -85,B 0,C 180,E1 -7082.706,E2 -7082.706} C_VEL
LIN {X 0,Y 477.64,Z 657.787,A -85,B 0,C 180,E1 -7082.77,E2 -7082.77} C_VEL
LIN {X 0,Y 477.441,Z 678.062,A -85,B 0,C 180,E1 -7083.117,E2 -7083.117} C_VEL
LIN {X 0,Y 477.292,Z 690.124,A -85,B 0,C 180,E1 -7083.491,E2 -7083.491} C_VEL
LIN {X 0,Y 476.96,Z 703.027,A -85,B 0,C 180,E1 -7084.068,E2 -7084.068} C_VEL
LIN {X 0,Y 476.533,Z 715.064,A -85,B 0,C 180,E1 -7084.796,E2 -7084.796} C_VEL
LIN {X 0,Y 476.037,Z 726.551,A -85,B 0,C 180,E1 -7085.696,E2 -7085.696} C_VEL
LIN {X 0,Y 475.578,Z 736.913,A -85,B 0,C 180,E1 -7086.716,E2 -7086.716} C_VEL
LIN {X 0,Y 475.157,Z 746.092,A -85,B 0,C 180,E1 -7087.842,E2 -7087.842} C_VEL
LIN {X 0,Y 474.794,Z 753.487,A -85,B 0,C 180,E1 -7088.948,E2 -7088.948} C_VEL
LIN {X 0,Y 474.461,Z 760.867,A -85,B 0,C 180,E1 -7090.307,E2 -7090.307} C_VEL
LIN {X 0,Y 474.265,Z 766.082,A -85,B 0,C 180,E1 -7091.514,E2 -7091.514} C_VEL
LIN {X 0,Y 474.094,Z 770.335,A -85,B 0,C 180,E1 -7092.754,E2 -7092.754} C_VEL
LIN {X 0,Y 474.006,Z 772.725,A -85,B 0,C 180,E1 -7093.638,E2 -7093.638} C_VEL
LIN {X 0,Y 473.93,Z 774.737,A -85,B 0,C 180,E1 -7094.558,E2 -7094.558} C_VEL
LIN {X 0,Y 473.855,Z 776.156,A -85,B 0,C 180,E1 -7095.396,E2 -7095.396} C_VEL
LIN {X 0,Y 473.799,Z 777.803,A -85,B 0,C 180,E1 -7097.144,E2 -7097.144} C_VEL
LIN {X 0,Y 473.838,Z 778.008,A -85,B 0,C 180,E1 -7098.215,E2 -7098.215} C_VEL
LIN {X 0,Y 473.821,Z 777.219,A -85,B 0,C 180,E1 -7099.747,E2 -7099.747} C_VEL
LIN {X 0,Y 473.843,Z 776.229,A -85,B 0,C 180,E1 -7100.61,E2 -7100.61} C_VEL
LIN {X 0,Y 473.896,Z 774.817,A -85,B 0,C 180,E1 -7101.472,E2 -7101.472} C_VEL
LIN {X 0,Y 474.094,Z 771.882,A -85,B 0,C 180,E1 -7102.761,E2 -7102.761} C_VEL
LIN {X 0,Y 474.15,Z 767.946,A -85,B 0,C 180,E1 -7104.045,E2 -7104.045} C_VEL
LIN {X 0,Y 474.336,Z 762.864,A -85,B 0,C 180,E1 -7105.326,E2 -7105.326} C_VEL
LIN {X 0,Y 474.62,Z 756.489,A -85,B 0,C 180,E1 -7106.604,E2 -7106.604} C_VEL
LIN {X 0,Y 474.964,Z 748.597,A -85,B 0,C 180,E1 -7107.88,E2 -7107.88} C_VEL
LIN {X 0,Y 475.409,Z 740.507,A -85,B 0,C 180,E1 -7108.941,E2 -7108.941} C_VEL
LIN {X 0,Y 475.819,Z 730.611,A -85,B 0,C 180,E1 -7110,E2 -7110} C_VEL
LIN {X 0,Y 476.264,Z 719.566,A -85,B 0,C 180,E1 -7110.951,E2 -7110.951} C_VEL
LIN {X 0,Y 476.763,Z 708.652,A -85,B 0,C 180,E1 -7111.689,E2 -7111.689} C_VEL
LIN {X 0,Y 477.079,Z 696.499,A -85,B 0,C 180,E1 -7112.322,E2 -7112.322} C_VEL
LIN {X 0,Y 477.364,Z 683.922,A -85,B 0,C 180,E1 -7112.795,E2 -7112.795} C_VEL
LIN {X 0,Y 477.564,Z 670.542,A -85,B 0,C 180,E1 -7113.111,E2 -7113.111} C_VEL
LIN {X 0,Y 478.082,Z 581.202,A -85,B 0,C 180,E1 -7114.465,E2 -7114.465} C_VEL
LIN {X 0,Y 474.697,Z 571.355,A -85,B 0,C 180,E1 -7114.75,E2 -7114.75} C_VEL
LIN {X 0,Y 474.763,Z 571.345,A -85,B 0,C 180,E1 -7117.335,E2 -7117.335} C_VEL
LIN {X 0,Y 474.682,Z 571.358,A -85,B 0,C 180,E1 -7120.234,E2 -7120.234} C_VEL
LIN {X 0,Y 474.681,Z 571.353,A -85,B 0,C 180,E1 -7122.831,E2 -7122.831} C_VEL
LIN {X 0,Y 474.683,Z 571.357,A -85,B 0,C 180,E1 -7125.768,E2 -7125.768} C_VEL
LIN {X 0,Y 474.666,Z 571.354,A -85,B 0,C 180,E1 -7129.01,E2 -7129.01} C_VEL
LIN {X 0,Y 474.59,Z 571.367,A -85,B 0,C 180,E1 -7131.728,E2 -7131.728} C_VEL
LIN {X 0,Y 474.639,Z 571.361,A -85,B 0,C 180,E1 -7134.493,E2 -7134.493} C_VEL
LIN {X 0,Y 474.699,Z 571.353,A -85,B 0,C 180,E1 -7137.338,E2 -7137.338} C_VEL
LIN {X 0,Y 474.662,Z 571.36,A -85,B 0,C 180,E1 -7139.326,E2 -7139.326} C_VEL
LIN {X 0,Y 478.199,Z 581.429,A -85,B 0,C 180,E1 -7139.629,E2 -7139.629} C_VEL
LIN {X 0,Y 477.38,Z 675.146,A -85,B 0,C 180,E1 -7141.095,E2 -7141.095} C_VEL
LIN {X 0,Y 477.233,Z 688.653,A -85,B 0,C 180,E1 -7141.487,E2 -7141.487} C_VEL
LIN {X 0,Y 476.913,Z 701.493,A -85,B 0,C 180,E1 -7142.039,E2 -7142.039} C_VEL
LIN {X 0,Y 476.479,Z 714.01,A -85,B 0,C 180,E1 -7142.781,E2 -7142.781} C_VEL
LIN {X 0,Y 476.044,Z 724.971,A -85,B 0,C 180,E1 -7143.615,E2 -7143.615} C_VEL
LIN {X 0,Y 475.647,Z 734.765,A -85,B 0,C 180,E1 -7144.541,E2 -7144.541} C_VEL
LIN {X 0,Y 475.168,Z 744.54,A -85,B 0,C 180,E1 -7145.688,E2 -7145.688} C_VEL
LIN {X 0,Y 474.8,Z 753.113,A -85,B 0,C 180,E1 -7146.936,E2 -7146.936} C_VEL
LIN {X 0,Y 474.475,Z 760.492,A -85,B 0,C 180,E1 -7148.275,E2 -7148.275} C_VEL
LIN {X 0,Y 474.273,Z 766.226,A -85,B 0,C 180,E1 -7149.596,E2 -7149.596} C_VEL
LIN {X 0,Y 474.052,Z 770.605,A -85,B 0,C 180,E1 -7150.879,E2 -7150.879} C_VEL
LIN {X 0,Y 473.932,Z 773.871,A -85,B 0,C 180,E1 -7152.144,E2 -7152.144} C_VEL
LIN {X 0,Y 473.835,Z 776.153,A -85,B 0,C 180,E1 -7153.383,E2 -7153.383} C_VEL
LIN {X 0,Y 473.782,Z 777.538,A -85,B 0,C 180,E1 -7154.6,E2 -7154.6} C_VEL
LIN {X 0,Y 473.725,Z 778.096,A -85,B 0,C 180,E1 -7155.791,E2 -7155.791} C_VEL
LIN {X 0,Y 473.771,Z 777.9,A -85,B 0,C 180,E1 -7156.971,E2 -7156.971} C_VEL
LIN {X 0,Y 473.815,Z 776.995,A -85,B 0,C 180,E1 -7158.127,E2 -7158.127} C_VEL
LIN {X 0,Y 473.903,Z 774.264,A -85,B 0,C 180,E1 -7159.826,E2 -7159.826} C_VEL
LIN {X 0,Y 474.138,Z 769.929,A -85,B 0,C 180,E1 -7161.497,E2 -7161.497} C_VEL
LIN {X 0,Y 474.343,Z 764.846,A -85,B 0,C 180,E1 -7162.9,E2 -7162.9} C_VEL
LIN {X 0,Y 474.619,Z 757.954,A -85,B 0,C 180,E1 -7164.369,E2 -7164.369} C_VEL
LIN {X 0,Y 474.89,Z 751.152,A -85,B 0,C 180,E1 -7165.523,E2 -7165.523} C_VEL
LIN {X 0,Y 475.362,Z 742.51,A -85,B 0,C 180,E1 -7166.71,E2 -7166.71} C_VEL
LIN {X 0,Y 475.727,Z 733.759,A -85,B 0,C 180,E1 -7167.696,E2 -7167.696} C_VEL
LIN {X 0,Y 476.191,Z 723.047,A -85,B 0,C 180,E1 -7168.676,E2 -7168.676} C_VEL
LIN {X 0,Y 476.609,Z 711.975,A -85,B 0,C 180,E1 -7169.482,E2 -7169.482} C_VEL
LIN {X 0,Y 476.993,Z 700.468,A -85,B 0,C 180,E1 -7170.127,E2 -7170.127} C_VEL
LIN {X 0,Y 477.221,Z 687.353,A -85,B 0,C 180,E1 -7170.673,E2 -7170.673} C_VEL
LIN {X 0,Y 477.457,Z 674.525,A -85,B 0,C 180,E1 -7171.021,E2 -7171.021} C_VEL
LIN {X 0,Y 478.177,Z 581.442,A -85,B 0,C 180,E1 -7172.48,E2 -7172.48} C_VEL
LIN {X 0,Y 474.712,Z 571.356,A -85,B 0,C 180,E1 -7172.79,E2 -7172.79} C_VEL
LIN {X 0,Y 474.651,Z 571.359,A -85,B 0,C 180,E1 -7175.507,E2 -7175.507} C_VEL
LIN {X 0,Y 474.661,Z 571.358,A -85,B 0,C 180,E1 -7179.185,E2 -7179.185} C_VEL
LIN {X 0,Y 474.648,Z 571.359,A -85,B 0,C 180,E1 -7181.884,E2 -7181.884} C_VEL
LIN {X 0,Y 474.69,Z 571.359,A -85,B 0,C 180,E1 -7184.544,E2 -7184.544} C_VEL
LIN {X 0,Y 474.729,Z 571.35,A -85,B 0,C 180,E1 -7188.038,E2 -7188.038} C_VEL
LIN {X 0,Y 474.719,Z 571.349,A -85,B 0,C 180,E1 -7191.486,E2 -7191.486} C_VEL
LIN {X 0,Y 474.78,Z 571.344,A -85,B 0,C 180,E1 -7194.052,E2 -7194.052} C_VEL
LIN {X 0,Y 474.886,Z 571.326,A -85,B 0,C 180,E1 -7197.455,E2 -7197.455} C_VEL
LIN {X 0,Y 474.867,Z 571.334,A -85,B 0,C 180,E1 -7200.848,E2 -7200.848} C_VEL
LIN {X 0,Y 474.885,Z 571.333,A -85,B 0,C 180,E1 -7202.545,E2 -7202.545} C_VEL
LIN {X 0,Y 474.781,Z 571.341,A -85,B 0,C 180,E1 -7205.948,E2 -7205.948} C_VEL
LIN {X 0,Y 474.719,Z 571.354,A -85,B 0,C 180,E1 -7208.514,E2 -7208.514} C_VEL
LIN {X 0,Y 474.729,Z 571.346,A -85,B 0,C 180,E1 -7211.962,E2 -7211.962} C_VEL
LIN {X 0,Y 474.671,Z 571.352,A -85,B 0,C 180,E1 -7215.768,E2 -7215.768} C_VEL
LIN {X 0,Y 474.656,Z 571.355,A -85,B 0,C 180,E1 -7219.011,E2 -7219.011} C_VEL
LIN {X 0,Y 474.589,Z 571.363,A -85,B 0,C 180,E1 -7221.729,E2 -7221.729} C_VEL
LIN {X 0,Y 474.654,Z 571.36,A -85,B 0,C 180,E1 -7224.493,E2 -7224.493} C_VEL
LIN {X 0,Y 474.691,Z 571.349,A -85,B 0,C 180,E1 -7227.339,E2 -7227.339} C_VEL
LIN {X 0,Y 474.603,Z 571.366,A -85,B 0,C 180,E1 -7230.812,E2 -7230.812} C_VEL
LIN {X 0,Y 474.632,Z 571.359,A -85,B 0,C 180,E1 -7233.985,E2 -7233.985} C_VEL
LIN {X 0,Y 474.57,Z 571.37,A -85,B 0,C 180,E1 -7236.901,E2 -7236.901} C_VEL
LIN {X 0,Y 474.649,Z 571.356,A -85,B 0,C 180,E1 -7239.652,E2 -7239.652} C_VEL
LIN {X 0,Y 474.647,Z 571.36,A -85,B 0,C 180,E1 -7242.931,E2 -7242.931} C_VEL
LIN {X 0,Y 474.605,Z 571.365,A -85,B 0,C 180,E1 -7245.896,E2 -7245.896} C_VEL
LIN {X 0,Y 474.636,Z 571.36,A -85,B 0,C 180,E1 -7249.04,E2 -7249.04} C_VEL
LIN {X 0,Y 474.614,Z 571.363,A -85,B 0,C 180,E1 -7251.704,E2 -7251.704} C_VEL
LIN {X 0,Y 474.624,Z 571.364,A -85,B 0,C 180,E1 -7254.727,E2 -7254.727} C_VEL
LIN {X 0,Y 474.635,Z 571.362,A -85,B 0,C 180,E1 -7257.789,E2 -7257.789} C_VEL
LIN {X 0,Y 474.623,Z 571.366,A -85,B 0,C 180,E1 -7260.885,E2 -7260.885} C_VEL
LIN {X 0,Y 474.672,Z 571.434,A -85,B 0,C 180,E1 -7261.971,E2 -7261.971} C_VEL
LIN {X 0,Y 477.267,Z 584.263,A -85,B 0,C 180,E1 -7264.111,E2 -7264.111} C_VEL
LIN {X 0,Y 477.507,Z 588.241,A -85,B 0,C 180,E1 -7264.734,E2 -7264.734} C_VEL
LIN {X 0,Y 476.661,Z 607.871,A -85,B 0,C 180,E1 -7267.688,E2 -7267.688} C_VEL
LIN {X 0,Y 475.876,Z 629.113,A -85,B 0,C 180,E1 -7270.839,E2 -7270.839} C_VEL
LIN {X 0,Y 475.378,Z 645.48,A -85,B 0,C 180,E1 -7273.229,E2 -7273.229} C_VEL
LIN {X 0,Y 477.968,Z 666.813,A -85,B 0,C 180,E1 -7273.657,E2 -7273.657} C_VEL
LIN {X 0,Y 477.231,Z 755.411,A -85,B 0,C 180,E1 -7275.039,E2 -7275.039} C_VEL
LIN {X 0,Y 476.849,Z 769.349,A -85,B 0,C 180,E1 -7275.436,E2 -7275.436} C_VEL
LIN {X 0,Y 476.452,Z 781.893,A -85,B 0,C 180,E1 -7275.968,E2 -7275.968} C_VEL
LIN {X 0,Y 475.987,Z 793.915,A -85,B 0,C 180,E1 -7276.662,E2 -7276.662} C_VEL
LIN {X 0,Y 475.539,Z 805.757,A -85,B 0,C 180,E1 -7277.541,E2 -7277.541} C_VEL
LIN {X 0,Y 475.004,Z 815.907,A -85,B 0,C 180,E1 -7278.478,E2 -7278.478} C_VEL
LIN {X 0,Y 474.647,Z 825.301,A -85,B 0,C 180,E1 -7279.55,E2 -7279.55} C_VEL
LIN {X 0,Y 474.308,Z 834.444,A -85,B 0,C 180,E1 -7280.835,E2 -7280.835} C_VEL
LIN {X 0,Y 474.073,Z 841.819,A -85,B 0,C 180,E1 -7282.118,E2 -7282.118} C_VEL
LIN {X 0,Y 473.893,Z 848.223,A -85,B 0,C 180,E1 -7283.533,E2 -7283.533} C_VEL
LIN {X 0,Y 473.847,Z 852.999,A -85,B 0,C 180,E1 -7284.895,E2 -7284.895} C_VEL
LIN {X 0,Y 473.838,Z 855.365,A -85,B 0,C 180,E1 -7285.747,E2 -7285.747} C_VEL
LIN {X 0,Y 473.835,Z 857.286,A -85,B 0,C 180,E1 -7286.599,E2 -7286.599} C_VEL
LIN {X 0,Y 473.864,Z 858.728,A -85,B 0,C 180,E1 -7287.45,E2 -7287.45} C_VEL
LIN {X 0,Y 473.707,Z 860.381,A -85,B 0,C 180,E1 -7289.15,E2 -7289.15} C_VEL
LIN {X 0,Y 473.702,Z 860.614,A -85,B 0,C 180,E1 -7290,E2 -7290} C_VEL
LIN {X 0,Y 473.761,Z 859.798,A -85,B 0,C 180,E1 -7291.7,E2 -7291.7} C_VEL
LIN {X 0,Y 473.864,Z 858.801,A -85,B 0,C 180,E1 -7292.55,E2 -7292.55} C_VEL
LIN {X 0,Y 473.832,Z 857.38,A -85,B 0,C 180,E1 -7293.401,E2 -7293.401} C_VEL
LIN {X 0,Y 473.789,Z 854.396,A -85,B 0,C 180,E1 -7294.68,E2 -7294.68} C_VEL
LIN {X 0,Y 473.879,Z 850.362,A -85,B 0,C 180,E1 -7295.959,E2 -7295.959} C_VEL
LIN {X 0,Y 474.017,Z 844.14,A -85,B 0,C 180,E1 -7297.454,E2 -7297.454} C_VEL
LIN {X 0,Y 474.221,Z 837.354,A -85,B 0,C 180,E1 -7298.737,E2 -7298.737} C_VEL
LIN {X 0,Y 474.509,Z 828.94,A -85,B 0,C 180,E1 -7300.022,E2 -7300.022} C_VEL
LIN {X 0,Y 474.902,Z 820.3,A -85,B 0,C 180,E1 -7301.092,E2 -7301.092} C_VEL
LIN {X 0,Y 475.339,Z 810.092,A -85,B 0,C 180,E1 -7302.122,E2 -7302.122} C_VEL
LIN {X 0,Y 475.753,Z 799.098,A -85,B 0,C 180,E1 -7303.019,E2 -7303.019} C_VEL
LIN {X 0,Y 476.238,Z 787.511,A -85,B 0,C 180,E1 -7303.766,E2 -7303.766} C_VEL
LIN {X 0,Y 476.71,Z 775.516,A -85,B 0,C 180,E1 -7304.351,E2 -7304.351} C_VEL
LIN {X 0,Y 477.065,Z 762.57,A -85,B 0,C 180,E1 -7304.803,E2 -7304.803} C_VEL
LIN {X 0,Y 477.365,Z 748.914,A -85,B 0,C 180,E1 -7305.094,E2 -7305.094} C_VEL
LIN {X 0,Y 477.883,Z 662.522,A -85,B 0,C 180,E1 -7306.426,E2 -7306.426} C_VEL
LIN {X 0,Y 475.765,Z 645.286,A -85,B 0,C 180,E1 -7306.785,E2 -7306.785} C_VEL
LIN {X 0,Y 476.656,Z 619.964,A -85,B 0,C 180,E1 -7310.047,E2 -7310.047} C_VEL
LIN {X 0,Y 477.719,Z 594.261,A -85,B 0,C 180,E1 -7313.403,E2 -7313.403} C_VEL
LIN {X 0,Y 478.017,Z 587.403,A -85,B 0,C 180,E1 -7314.309,E2 -7314.309} C_VEL
LIN {X 0,Y 475.443,Z 574.636,A -85,B 0,C 180,E1 -7316.153,E2 -7316.153} C_VEL
LIN {X 0,Y 474.713,Z 571.354,A -85,B 0,C 180,E1 -7316.664,E2 -7316.664} C_VEL
LIN {X 0,Y 474.621,Z 571.364,A -85,B 0,C 180,E1 -7319.251,E2 -7319.251} C_VEL
LIN {X 0,Y 474.615,Z 571.364,A -85,B 0,C 180,E1 -7322.43,E2 -7322.43} C_VEL
LIN {X 0,Y 474.619,Z 571.363,A -85,B 0,C 180,E1 -7325.469,E2 -7325.469} C_VEL
LIN {X 0,Y 474.62,Z 571.362,A -85,B 0,C 180,E1 -7328.455,E2 -7328.455} C_VEL
LIN {X 0,Y 474.638,Z 571.357,A -85,B 0,C 180,E1 -7330.96,E2 -7330.96} C_VEL
LIN {X 0,Y 474.605,Z 571.37,A -85,B 0,C 180,E1 -7334.104,E2 -7334.104} C_VEL
LIN {X 0,Y 474.647,Z 571.356,A -85,B 0,C 180,E1 -7337.069,E2 -7337.069} C_VEL
LIN {X 0,Y 474.668,Z 571.356,A -85,B 0,C 180,E1 -7340.456,E2 -7340.456} C_VEL
LIN {X 0,Y 474.587,Z 571.365,A -85,B 0,C 180,E1 -7343.676,E2 -7343.676} C_VEL
LIN {X 0,Y 474.636,Z 571.359,A -85,B 0,C 180,E1 -7346.779,E2 -7346.779} C_VEL
LIN {X 0,Y 474.606,Z 571.362,A -85,B 0,C 180,E1 -7349.77,E2 -7349.77} C_VEL
LIN {X 0,Y 474.707,Z 571.353,A -85,B 0,C 180,E1 -7352.68,E2 -7352.68} C_VEL
LIN {X 0,Y 474.651,Z 571.355,A -85,B 0,C 180,E1 -7355.507,E2 -7355.507} C_VEL
LIN {X 0,Y 474.661,Z 571.354,A -85,B 0,C 180,E1 -7359.185,E2 -7359.185} C_VEL
LIN {X 0,Y 474.648,Z 571.357,A -85,B 0,C 180,E1 -7361.884,E2 -7361.884} C_VEL
LIN {X 0,Y 474.69,Z 571.349,A -85,B 0,C 180,E1 -7364.544,E2 -7364.544} C_VEL
LIN {X 0,Y 474.695,Z 571.352,A -85,B 0,C 180,E1 -7368.037,E2 -7368.037} C_VEL
LIN {X 0,Y 474.719,Z 571.339,A -85,B 0,C 180,E1 -7371.486,E2 -7371.486} C_VEL
LIN {X 0,Y 474.782,Z 571.34,A -85,B 0,C 180,E1 -7374.052,E2 -7374.052} C_VEL
LIN {X 0,Y 474.886,Z 571.32,A -85,B 0,C 180,E1 -7377.455,E2 -7377.455} C_VEL
LIN {X 0,Y 474.867,Z 571.336,A -85,B 0,C 180,E1 -7380.848,E2 -7380.848} C_VEL
LIN {X 0,Y 474.885,Z 571.333,A -85,B 0,C 180,E1 -7382.545,E2 -7382.545} C_VEL
LIN {X 0,Y 474.776,Z 571.331,A -85,B 0,C 180,E1 -7385.948,E2 -7385.948} C_VEL
LIN {X 0,Y 474.719,Z 571.35,A -85,B 0,C 180,E1 -7388.514,E2 -7388.514} C_VEL
LIN {X 0,Y 474.695,Z 571.344,A -85,B 0,C 180,E1 -7391.963,E2 -7391.963} C_VEL
LIN {X 0,Y 474.69,Z 571.353,A -85,B 0,C 180,E1 -7395.456,E2 -7395.456} C_VEL
LIN {X 0,Y 474.656,Z 571.355,A -85,B 0,C 180,E1 -7399.011,E2 -7399.011} C_VEL
LIN {X 0,Y 474.579,Z 571.366,A -85,B 0,C 180,E1 -7401.729,E2 -7401.729} C_VEL
LIN {X 0,Y 474.65,Z 571.354,A -85,B 0,C 180,E1 -7404.493,E2 -7404.493} C_VEL
LIN {X 0,Y 474.691,Z 571.356,A -85,B 0,C 180,E1 -7407.339,E2 -7407.339} C_VEL
LIN {X 0,Y 474.61,Z 571.361,A -85,B 0,C 180,E1 -7410.813,E2 -7410.813} C_VEL
LIN {X 0,Y 474.631,Z 571.355,A -85,B 0,C 180,E1 -7413.985,E2 -7413.985} C_VEL
LIN {X 0,Y 474.57,Z 571.371,A -85,B 0,C 180,E1 -7416.901,E2 -7416.901} C_VEL
LIN {X 0,Y 474.638,Z 571.358,A -85,B 0,C 180,E1 -7419.651,E2 -7419.651} C_VEL
LIN {X 0,Y 474.63,Z 571.349,A -85,B 0,C 180,E1 -7422.933,E2 -7422.933} C_VEL
LIN {X 0,Y 474.603,Z 571.362,A -85,B 0,C 180,E1 -7425.896,E2 -7425.896} C_VEL
LIN {X 0,Y 474.624,Z 571.359,A -85,B 0,C 180,E1 -7429.042,E2 -7429.042} C_VEL
LIN {X 0,Y 474.608,Z 571.36,A -85,B 0,C 180,E1 -7431.705,E2 -7431.705} C_VEL
LIN {X 0,Y 474.628,Z 571.36,A -85,B 0,C 180,E1 -7434.727,E2 -7434.727} C_VEL
LIN {X 0,Y 474.635,Z 571.363,A -85,B 0,C 180,E1 -7437.789,E2 -7437.789} C_VEL
LIN {X 0,Y 474.678,Z 571.359,A -85,B 0,C 180,E1 -7441.313,E2 -7441.313} C_VEL
LIN {X 0,Y 478.196,Z 581.606,A -85,B 0,C 180,E1 -7441.617,E2 -7441.617} C_VEL
LIN {X 0,Y 477.64,Z 657.787,A -85,B 0,C 180,E1 -7442.77,E2 -7442.77} C_VEL
LIN {X 0,Y 476.857,Z 663.642,A -85,B 0,C 180,E1 -7442.829,E2 -7442.829} C_VEL
LIN {X 0,Y 473.858,Z 673.131,A -85,B 0,C 180,E1 -7442.881,E2 -7442.881} C_VEL
LIN {X 0,Y 471.037,Z 682.595,A -85,B 0,C 180,E1 -7443.012,E2 -7443.012} C_VEL
LIN {X 0,Y 470.478,Z 688.236,A -85,B 0,C 180,E1 -7443.175,E2 -7443.175} C_VEL
LIN {X 0,Y 470.227,Z 700.368,A -85,B 0,C 180,E1 -7443.684,E2 -7443.684} C_VEL
LIN {X 0,Y 469.79,Z 712.951,A -85,B 0,C 180,E1 -7444.408,E2 -7444.408} C_VEL
LIN {X 0,Y 469.35,Z 723.78,A -85,B 0,C 180,E1 -7445.212,E2 -7445.212} C_VEL
LIN {X 0,Y 468.844,Z 733.655,A -85,B 0,C 180,E1 -7446.126,E2 -7446.126} C_VEL
LIN {X 0,Y 468.38,Z 743.595,A -85,B 0,C 180,E1 -7447.271,E2 -7447.271} C_VEL
LIN {X 0,Y 467.979,Z 751.316,A -85,B 0,C 180,E1 -7448.359,E2 -7448.359} C_VEL
LIN {X 0,Y 467.637,Z 758.274,A -85,B 0,C 180,E1 -7449.549,E2 -7449.549} C_VEL
LIN {X 0,Y 467.366,Z 763.701,A -85,B 0,C 180,E1 -7450.682,E2 -7450.682} C_VEL
LIN {X 0,Y 467.16,Z 768.931,A -85,B 0,C 180,E1 -7452.037,E2 -7452.037} C_VEL
LIN {X 0,Y 466.985,Z 772.896,A -85,B 0,C 180,E1 -7453.385,E2 -7453.385} C_VEL
LIN {X 0,Y 466.889,Z 775.231,A -85,B 0,C 180,E1 -7454.447,E2 -7454.447} C_VEL
LIN {X 0,Y 466.73,Z 777.622,A -85,B 0,C 180,E1 -7456.059,E2 -7456.059} C_VEL
LIN {X 0,Y 466.735,Z 778.607,A -85,B 0,C 180,E1 -7457.831,E2 -7457.831} C_VEL
LIN {X 0,Y 466.763,Z 778.513,A -85,B 0,C 180,E1 -7458.712,E2 -7458.712} C_VEL
LIN {X 0,Y 466.769,Z 777.98,A -85,B 0,C 180,E1 -7459.591,E2 -7459.591} C_VEL
LIN {X 0,Y 466.838,Z 775.739,A -85,B 0,C 180,E1 -7461.342,E2 -7461.342} C_VEL
LIN {X 0,Y 467.002,Z 772.939,A -85,B 0,C 180,E1 -7462.651,E2 -7462.651} C_VEL
LIN {X 0,Y 467.1,Z 769.144,A -85,B 0,C 180,E1 -7463.954,E2 -7463.954} C_VEL
LIN {X 0,Y 467.293,Z 764.236,A -85,B 0,C 180,E1 -7465.255,E2 -7465.255} C_VEL
LIN {X 0,Y 467.585,Z 758.039,A -85,B 0,C 180,E1 -7466.553,E2 -7466.553} C_VEL
LIN {X 0,Y 467.915,Z 750.34,A -85,B 0,C 180,E1 -7467.848,E2 -7467.848} C_VEL
LIN {X 0,Y 468.352,Z 742.482,A -85,B 0,C 180,E1 -7468.925,E2 -7468.925} C_VEL
LIN {X 0,Y 468.813,Z 732.96,A -85,B 0,C 180,E1 -7470,E2 -7470} C_VEL
LIN {X 0,Y 469.233,Z 722.298,A -85,B 0,C 180,E1 -7470.965,E2 -7470.965} C_VEL
LIN {X 0,Y 469.844,Z 710.245,A -85,B 0,C 180,E1 -7471.821,E2 -7471.821} C_VEL
LIN {X 0,Y 470.187,Z 698.445,A -85,B 0,C 180,E1 -7472.463,E2 -7472.463} C_VEL
LIN {X 0,Y 470.484,Z 685.556,A -85,B 0,C 180,E1 -7472.97,E2 -7472.97} C_VEL
LIN {X 0,Y 470.687,Z 673.099,A -85,B 0,C 180,E1 -7473.29,E2 -7473.29} C_VEL
LIN {X 0,Y 471.338,Z 583.023,A -85,B 0,C 180,E1 -7474.676,E2 -7474.676} C_VEL
LIN {X 0,Y 467.684,Z 572.228,A -85,B 0,C 180,E1 -7474.984,E2 -7474.984} C_VEL
LIN {X 0,Y 467.696,Z 572.229,A -85,B 0,C 180,E1 -7477.772,E2 -7477.772} C_VEL
LIN {X 0,Y 467.673,Z 572.226,A -85,B 0,C 180,E1 -7481.265,E2 -7481.265} C_VEL
LIN {X 0,Y 467.613,Z 572.239,A -85,B 0,C 180,E1 -7483.914,E2 -7483.914} C_VEL
LIN {X 0,Y 467.599,Z 572.237,A -85,B 0,C 180,E1 -7486.592,E2 -7486.592} C_VEL
LIN {X 0,Y 467.625,Z 572.232,A -85,B 0,C 180,E1 -7489.307,E2 -7489.307} C_VEL
LIN {X 0,Y 467.536,Z 572.25,A -85,B 0,C 180,E1 -7492.073,E2 -7492.073} C_VEL
LIN {X 0,Y 467.585,Z 572.237,A -85,B 0,C 180,E1 -7494.888,E2 -7494.888} C_VEL
LIN {X 0,Y 467.628,Z 572.238,A -85,B 0,C 180,E1 -7497.768,E2 -7497.768} C_VEL
LIN {X 0,Y 467.636,Z 572.234,A -85,B 0,C 180,E1 -7499.068,E2 -7499.068} C_VEL
LIN {X 0,Y 470.678,Z 580.961,A -85,B 0,C 180,E1 -7499.345,E2 -7499.345} C_VEL
LIN {X 0,Y 471.428,Z 583.273,A -85,B 0,C 180,E1 -7499.41,E2 -7499.41} C_VEL
LIN {X 0,Y 470.53,Z 676.185,A -85,B 0,C 180,E1 -7500.892,E2 -7500.892} C_VEL
LIN {X 0,Y 470.341,Z 689.732,A -85,B 0,C 180,E1 -7501.297,E2 -7501.297} C_VEL
LIN {X 0,Y 470.051,Z 701.678,A -85,B 0,C 180,E1 -7501.819,E2 -7501.819} C_VEL
LIN {X 0,Y 469.612,Z 713.669,A -85,B 0,C 180,E1 -7502.528,E2 -7502.528} C_VEL
LIN {X 0,Y 469.191,Z 724.651,A -85,B 0,C 180,E1 -7503.363,E2 -7503.363} C_VEL
LIN {X 0,Y 468.723,Z 735.137,A -85,B 0,C 180,E1 -7504.355,E2 -7504.355} C_VEL
LIN {X 0,Y 468.245,Z 744.283,A -85,B 0,C 180,E1 -7505.428,E2 -7505.428} C_VEL
LIN {X 0,Y 467.852,Z 752.812,A -85,B 0,C 180,E1 -7506.663,E2 -7506.663} C_VEL
LIN {X 0,Y 467.476,Z 760.54,A -85,B 0,C 180,E1 -7508.052,E2 -7508.052} C_VEL
LIN {X 0,Y 467.217,Z 766.919,A -85,B 0,C 180,E1 -7509.529,E2 -7509.529} C_VEL
LIN {X 0,Y 467.028,Z 771.051,A -85,B 0,C 180,E1 -7510.752,E2 -7510.752} C_VEL
LIN {X 0,Y 466.904,Z 774.216,A -85,B 0,C 180,E1 -7511.965,E2 -7511.965} C_VEL
LIN {X 0,Y 466.82,Z 775.606,A -85,B 0,C 180,E1 -7512.645,E2 -7512.645} C_VEL
LIN {X 0,Y 466.754,Z 777.403,A -85,B 0,C 180,E1 -7513.837,E2 -7513.837} C_VEL
LIN {X 0,Y 466.689,Z 778.448,A -85,B 0,C 180,E1 -7515.054,E2 -7515.054} C_VEL
LIN {X 0,Y 466.692,Z 778.721,A -85,B 0,C 180,E1 -7516.288,E2 -7516.288} C_VEL
LIN {X 0,Y 466.729,Z 778.18,A -85,B 0,C 180,E1 -7517.546,E2 -7517.546} C_VEL
LIN {X 0,Y 466.768,Z 776.756,A -85,B 0,C 180,E1 -7518.835,E2 -7518.835} C_VEL
LIN {X 0,Y 466.882,Z 774.355,A -85,B 0,C 180,E1 -7520.146,E2 -7520.146} C_VEL
LIN {X 0,Y 467.099,Z 770.874,A -85,B 0,C 180,E1 -7521.479,E2 -7521.479} C_VEL
LIN {X 0,Y 467.314,Z 765.414,A -85,B 0,C 180,E1 -7523.018,E2 -7523.018} C_VEL
LIN {X 0,Y 467.622,Z 758.555,A -85,B 0,C 180,E1 -7524.499,E2 -7524.499} C_VEL
LIN {X 0,Y 467.92,Z 751.579,A -85,B 0,C 180,E1 -7525.696,E2 -7525.696} C_VEL
LIN {X 0,Y 468.359,Z 744.094,A -85,B 0,C 180,E1 -7526.75,E2 -7526.75} C_VEL
LIN {X 0,Y 468.805,Z 734.596,A -85,B 0,C 180,E1 -7527.846,E2 -7527.846} C_VEL
LIN {X 0,Y 469.293,Z 724.211,A -85,B 0,C 180,E1 -7528.816,E2 -7528.816} C_VEL
LIN {X 0,Y 469.697,Z 713.244,A -85,B 0,C 180,E1 -7529.637,E2 -7529.637} C_VEL
LIN {X 0,Y 470.122,Z 702.032,A -85,B 0,C 180,E1 -7530.288,E2 -7530.288} C_VEL
LIN {X 0,Y 470.377,Z 688.793,A -85,B 0,C 180,E1 -7530.857,E2 -7530.857} C_VEL
LIN {X 0,Y 470.642,Z 675.783,A -85,B 0,C 180,E1 -7531.226,E2 -7531.226} C_VEL
LIN {X 0,Y 471.449,Z 583.068,A -85,B 0,C 180,E1 -7532.709,E2 -7532.709} C_VEL
LIN {X 0,Y 467.68,Z 572.288,A -85,B 0,C 180,E1 -7533.035,E2 -7533.035} C_VEL
LIN {X 0,Y 467.584,Z 572.243,A -85,B 0,C 180,E1 -7536.467,E2 -7536.467} C_VEL
LIN {X 0,Y 467.615,Z 572.236,A -85,B 0,C 180,E1 -7539.777,E2 -7539.777} C_VEL
LIN {X 0,Y 467.6,Z 572.242,A -85,B 0,C 180,E1 -7542.506,E2 -7542.506} C_VEL
LIN {X 0,Y 467.597,Z 572.238,A -85,B 0,C 180,E1 -7545.196,E2 -7545.196} C_VEL
LIN {X 0,Y 467.687,Z 572.226,A -85,B 0,C 180,E1 -7547.855,E2 -7547.855} C_VEL
LIN {X 0,Y 467.673,Z 572.227,A -85,B 0,C 180,E1 -7551.357,E2 -7551.357} C_VEL
LIN {X 0,Y 467.742,Z 572.22,A -85,B 0,C 180,E1 -7553.963,E2 -7553.963} C_VEL
LIN {X 0,Y 467.851,Z 572.202,A -85,B 0,C 180,E1 -7557.417,E2 -7557.417} C_VEL
LIN {X 0,Y 467.872,Z 572.203,A -85,B 0,C 180,E1 -7560,E2 -7560} C_VEL
LIN {X 0,Y 467.851,Z 572.209,A -85,B 0,C 180,E1 -7562.583,E2 -7562.583} C_VEL
LIN {X 0,Y 467.744,Z 572.219,A -85,B 0,C 180,E1 -7566.037,E2 -7566.037} C_VEL
LIN {X 0,Y 467.673,Z 572.23,A -85,B 0,C 180,E1 -7568.643,E2 -7568.643} C_VEL
LIN {X 0,Y 467.673,Z 572.227,A -85,B 0,C 180,E1 -7572.145,E2 -7572.145} C_VEL
LIN {X 0,Y 467.64,Z 572.228,A -85,B 0,C 180,E1 -7575.886,E2 -7575.886} C_VEL
LIN {X 0,Y 467.615,Z 572.23,A -85,B 0,C 180,E1 -7579.308,E2 -7579.308} C_VEL
LIN {X 0,Y 467.534,Z 572.244,A -85,B 0,C 180,E1 -7582.074,E2 -7582.074} C_VEL
LIN {X 0,Y 467.597,Z 572.239,A -85,B 0,C 180,E1 -7584.888,E2 -7584.888} C_VEL
LIN {X 0,Y 467.621,Z 572.23,A -85,B 0,C 180,E1 -7587.769,E2 -7587.769} C_VEL
LIN {X 0,Y 467.565,Z 572.241,A -85,B 0,C 180,E1 -7591.047,E2 -7591.047} C_VEL
LIN {X 0,Y 467.583,Z 572.239,A -85,B 0,C 180,E1 -7594.243,E2 -7594.243} C_VEL
LIN {X 0,Y 467.546,Z 572.243,A -85,B 0,C 180,E1 -7597.188,E2 -7597.188} C_VEL
LIN {X 0,Y 467.592,Z 572.24,A -85,B 0,C 180,E1 -7600.263,E2 -7600.263} C_VEL
LIN {X 0,Y 467.614,Z 572.241,A -85,B 0,C 180,E1 -7602.572,E2 -7602.572} C_VEL
LIN {X 0,Y 467.566,Z 572.242,A -85,B 0,C 180,E1 -7605.054,E2 -7605.054} C_VEL
LIN {X 0,Y 467.585,Z 572.238,A -85,B 0,C 180,E1 -7607.441,E2 -7607.441} C_VEL
LIN {X 0,Y 467.613,Z 572.238,A -85,B 0,C 180,E1 -7610.859,E2 -7610.859} C_VEL
LIN {X 0,Y 467.558,Z 572.246,A -85,B 0,C 180,E1 -7614.262,E2 -7614.262} C_VEL
LIN {X 0,Y 467.58,Z 572.24,A -85,B 0,C 180,E1 -7617.322,E2 -7617.322} C_VEL
LIN {X 0,Y 467.569,Z 572.246,A -85,B 0,C 180,E1 -7620.668,E2 -7620.668} C_VEL
LIN {X 0,Y 467.629,Z 572.333,A -85,B 0,C 180,E1 -7621.745,E2 -7621.745} C_VEL
LIN {X 0,Y 470.239,Z 585.092,A -85,B 0,C 180,E1 -7623.914,E2 -7623.914} C_VEL
LIN {X 0,Y 470.595,Z 589.181,A -85,B 0,C 180,E1 -7624.574,E2 -7624.574} C_VEL
LIN {X 0,Y 469.692,Z 608.769,A -85,B 0,C 180,E1 -7627.57,E2 -7627.57} C_VEL
LIN {X 0,Y 468.86,Z 630.144,A -85,B 0,C 180,E1 -7630.794,E2 -7630.794} C_VEL
LIN {X 0,Y 468.321,Z 644.673,A -85,B 0,C 180,E1 -7632.96,E2 -7632.96} C_VEL
LIN {X 0,Y 471.13,Z 666.15,A -85,B 0,C 180,E1 -7633.413,E2 -7633.413} C_VEL
LIN {X 0,Y 470.373,Z 754.578,A -85,B 0,C 180,E1 -7634.815,E2 -7634.815} C_VEL
LIN {X 0,Y 470.002,Z 767.802,A -85,B 0,C 180,E1 -7635.191,E2 -7635.191} C_VEL
LIN {X 0,Y 469.505,Z 781.139,A -85,B 0,C 180,E1 -7635.756,E2 -7635.756} C_VEL
LIN {X 0,Y 469.033,Z 793.188,A -85,B 0,C 180,E1 -7636.46,E2 -7636.46} C_VEL
LIN {X 0,Y 468.567,Z 804.442,A -85,B 0,C 180,E1 -7637.302,E2 -7637.302} C_VEL
LIN {X 0,Y 468.031,Z 815.214,A -85,B 0,C 180,E1 -7638.304,E2 -7638.304} C_VEL
LIN {X 0,Y 467.614,Z 824.616,A -85,B 0,C 180,E1 -7639.391,E2 -7639.391} C_VEL
LIN {X 0,Y 467.244,Z 833.767,A -85,B 0,C 180,E1 -7640.695,E2 -7640.695} C_VEL
LIN {X 0,Y 467.02,Z 841.155,A -85,B 0,C 180,E1 -7641.999,E2 -7641.999} C_VEL
LIN {X 0,Y 466.912,Z 846.147,A -85,B 0,C 180,E1 -7643.084,E2 -7643.084} C_VEL
LIN {X 0,Y 466.845,Z 851.009,A -85,B 0,C 180,E1 -7644.385,E2 -7644.385} C_VEL
LIN {X 0,Y 466.741,Z 854.728,A -85,B 0,C 180,E1 -7645.682,E2 -7645.682} C_VEL
LIN {X 0,Y 466.766,Z 856.656,A -85,B 0,C 180,E1 -7646.547,E2 -7646.547} C_VEL
LIN {X 0,Y 466.805,Z 858.105,A -85,B 0,C 180,E1 -7647.411,E2 -7647.411} C_VEL
LIN {X 0,Y 466.637,Z 859.764,A -85,B 0,C 180,E1 -7649.137,E2 -7649.137} C_VEL
LIN {X 0,Y 466.629,Z 859.999,A -85,B 0,C 180,E1 -7650,E2 -7650} C_VEL
LIN {X 0,Y 466.698,Z 859.188,A -85,B 0,C 180,E1 -7651.726,E2 -7651.726} C_VEL
LIN {X 0,Y 466.805,Z 858.192,A -85,B 0,C 180,E1 -7652.589,E2 -7652.589} C_VEL
LIN {X 0,Y 466.763,Z 856.769,A -85,B 0,C 180,E1 -7653.453,E2 -7653.453} C_VEL
LIN {X 0,Y 466.714,Z 853.783,A -85,B 0,C 180,E1 -7654.751,E2 -7654.751} C_VEL
LIN {X 0,Y 466.785,Z 849.744,A -85,B 0,C 180,E1 -7656.05,E2 -7656.05} C_VEL
LIN {X 0,Y 466.928,Z 843.516,A -85,B 0,C 180,E1 -7657.568,E2 -7657.568} C_VEL
LIN {X 0,Y 467.148,Z 836.725,A -85,B 0,C 180,E1 -7658.871,E2 -7658.871} C_VEL
LIN {X 0,Y 467.475,Z 828.305,A -85,B 0,C 180,E1 -7660.174,E2 -7660.174} C_VEL
LIN {X 0,Y 467.911,Z 819.65,A -85,B 0,C 180,E1 -7661.26,E2 -7661.26} C_VEL
LIN {X 0,Y 468.34,Z 809.665,A -85,B 0,C 180,E1 -7662.283,E2 -7662.283} C_VEL
LIN {X 0,Y 468.729,Z 799.843,A -85,B 0,C 180,E1 -7663.107,E2 -7663.107} C_VEL
LIN {X 0,Y 469.235,Z 788.595,A -85,B 0,C 180,E1 -7663.865,E2 -7663.865} C_VEL
LIN {X 0,Y 469.769,Z 776.032,A -85,B 0,C 180,E1 -7664.512,E2 -7664.512} C_VEL
LIN {X 0,Y 470.174,Z 763.53,A -85,B 0,C 180,E1 -7664.97,E2 -7664.97} C_VEL
LIN {X 0,Y 470.481,Z 750.996,A -85,B 0,C 180,E1 -7665.264,E2 -7665.264} C_VEL
LIN {X 0,Y 471.085,Z 663.523,A -85,B 0,C 180,E1 -7666.643,E2 -7666.643} C_VEL
LIN {X 0,Y 468.778,Z 644.601,A -85,B 0,C 180,E1 -7667.055,E2 -7667.055} C_VEL
LIN {X 0,Y 469.73,Z 619.401,A -85,B 0,C 180,E1 -7670.356,E2 -7670.356} C_VEL
LIN {X 0,Y 470.801,Z 595.416,A -85,B 0,C 180,E1 -7673.535,E2 -7673.535} C_VEL
LIN {X 0,Y 471.063,Z 588.346,A -85,B 0,C 180,E1 -7674.482,E2 -7674.482} C_VEL
LIN {X 0,Y 468.123,Z 574.428,A -85,B 0,C 180,E1 -7676.538,E2 -7676.538} C_VEL
LIN {X 0,Y 467.703,Z 572.227,A -85,B 0,C 180,E1 -7676.906,E2 -7676.906} C_VEL
LIN {X 0,Y 467.568,Z 572.241,A -85,B 0,C 180,E1 -7680.733,E2 -7680.733} C_VEL
LIN {X 0,Y 467.586,Z 572.243,A -85,B 0,C 180,E1 -7683.787,E2 -7683.787} C_VEL
LIN {X 0,Y 467.549,Z 572.242,A -85,B 0,C 180,E1 -7687.186,E2 -7687.186} C_VEL
LIN {X 0,Y 467.592,Z 572.241,A -85,B 0,C 180,E1 -7690.262,E2 -7690.262} C_VEL
LIN {X 0,Y 467.582,Z 572.239,A -85,B 0,C 180,E1 -7692.566,E2 -7692.566} C_VEL
LIN {X 0,Y 467.566,Z 572.237,A -85,B 0,C 180,E1 -7695.052,E2 -7695.052} C_VEL
LIN {X 0,Y 467.62,Z 572.232,A -85,B 0,C 180,E1 -7697.443,E2 -7697.443} C_VEL
LIN {X 0,Y 467.613,Z 572.231,A -85,B 0,C 180,E1 -7700.858,E2 -7700.858} C_VEL
LIN {X 0,Y 467.557,Z 572.242,A -85,B 0,C 180,E1 -7704.26,E2 -7704.26} C_VEL
LIN {X 0,Y 467.575,Z 572.237,A -85,B 0,C 180,E1 -7707.32,E2 -7707.32} C_VEL
LIN {X 0,Y 467.57,Z 572.234,A -85,B 0,C 180,E1 -7710.665,E2 -7710.665} C_VEL
LIN {X 0,Y 467.619,Z 572.232,A -85,B 0,C 180,E1 -7713.2,E2 -7713.2} C_VEL
LIN {X 0,Y 467.584,Z 572.234,A -85,B 0,C 180,E1 -7716.468,E2 -7716.468} C_VEL
LIN {X 0,Y 467.615,Z 572.232,A -85,B 0,C 180,E1 -7719.777,E2 -7719.777} C_VEL
LIN {X 0,Y 467.6,Z 572.236,A -85,B 0,C 180,E1 -7722.506,E2 -7722.506} C_VEL
LIN {X 0,Y 467.596,Z 572.232,A -85,B 0,C 180,E1 -7725.196,E2 -7725.196} C_VEL
LIN {X 0,Y 467.647,Z 572.229,A -85,B 0,C 180,E1 -7727.854,E2 -7727.854} C_VEL
LIN {X 0,Y 467.673,Z 572.217,A -85,B 0,C 180,E1 -7731.357,E2 -7731.357} C_VEL
LIN {X 0,Y 467.744,Z 572.216,A -85,B 0,C 180,E1 -7733.963,E2 -7733.963} C_VEL
LIN {X 0,Y 467.851,Z 572.196,A -85,B 0,C 180,E1 -7737.417,E2 -7737.417} C_VEL
LIN {X 0,Y 467.872,Z 572.196,A -85,B 0,C 180,E1 -7740,E2 -7740} C_VEL
LIN {X 0,Y 467.851,Z 572.209,A -85,B 0,C 180,E1 -7742.583,E2 -7742.583} C_VEL
LIN {X 0,Y 467.739,Z 572.207,A -85,B 0,C 180,E1 -7746.037,E2 -7746.037} C_VEL
LIN {X 0,Y 467.673,Z 572.23,A -85,B 0,C 180,E1 -7748.643,E2 -7748.643} C_VEL
LIN {X 0,Y 467.647,Z 572.223,A -85,B 0,C 180,E1 -7752.146,E2 -7752.146} C_VEL
LIN {X 0,Y 467.629,Z 572.231,A -85,B 0,C 180,E1 -7755.695,E2 -7755.695} C_VEL
LIN {X 0,Y 467.608,Z 572.232,A -85,B 0,C 180,E1 -7758.765,E2 -7758.765} C_VEL
LIN {X 0,Y 467.571,Z 572.243,A -85,B 0,C 180,E1 -7761.269,E2 -7761.269} C_VEL
LIN {X 0,Y 467.564,Z 572.234,A -85,B 0,C 180,E1 -7763.944,E2 -7763.944} C_VEL
LIN {X 0,Y 467.62,Z 572.235,A -85,B 0,C 180,E1 -7766.8,E2 -7766.8} C_VEL
LIN {X 0,Y 467.581,Z 572.233,A -85,B 0,C 180,E1 -7769.736,E2 -7769.736} C_VEL
LIN {X 0,Y 467.577,Z 572.241,A -85,B 0,C 180,E1 -7772.759,E2 -7772.759} C_VEL
LIN {X 0,Y 467.55,Z 572.242,A -85,B 0,C 180,E1 -7775.89,E2 -7775.89} C_VEL
LIN {X 0,Y 467.587,Z 572.244,A -85,B 0,C 180,E1 -7779.144,E2 -7779.144} C_VEL
LIN {X 0,Y 467.581,Z 572.224,A -85,B 0,C 180,E1 -7782.568,E2 -7782.568} C_VEL
LIN {X 0,Y 467.566,Z 572.243,A -85,B 0,C 180,E1 -7785.054,E2 -7785.054} C_VEL
LIN {X 0,Y 467.585,Z 572.233,A -85,B 0,C 180,E1 -7787.441,E2 -7787.441} C_VEL
LIN {X 0,Y 467.579,Z 572.24,A -85,B 0,C 180,E1 -7790.856,E2 -7790.856} C_VEL
LIN {X 0,Y 467.561,Z 572.24,A -85,B 0,C 180,E1 -7794.261,E2 -7794.261} C_VEL
LIN {X 0,Y 467.58,Z 572.243,A -85,B 0,C 180,E1 -7797.322,E2 -7797.322} C_VEL
LIN {X 0,Y 467.569,Z 572.241,A -85,B 0,C 180,E1 -7800.668,E2 -7800.668} C_VEL
LIN {X 0,Y 467.631,Z 572.332,A -85,B 0,C 180,E1 -7801.053,E2 -7801.053} C_VEL
LIN {X 0,Y 471.451,Z 582.943,A -85,B 0,C 180,E1 -7801.376,E2 -7801.376} C_VEL
LIN {X 0,Y 470.735,Z 675.609,A -85,B 0,C 180,E1 -7802.823,E2 -7802.823} C_VEL
LIN {X 0,Y 470.478,Z 688.236,A -85,B 0,C 180,E1 -7803.175,E2 -7803.175} C_VEL
LIN {X 0,Y 469.826,Z 692.062,A -85,B 0,C 180,E1 -7803.289,E2 -7803.289} C_VEL
LIN {X 0,Y 466.912,Z 698.063,A -85,B 0,C 180,E1 -7803.439,E2 -7803.439} C_VEL
LIN {X 0,Y 463.938,Z 703.941,A -85,B 0,C 180,E1 -7803.632,E2 -7803.632} C_VEL
LIN {X 0,Y 463.193,Z 707.557,A -85,B 0,C 180,E1 -7803.815,E2 -7803.815} C_VEL
LIN {X 0,Y 462.701,Z 719.192,A -85,B 0,C 180,E1 -7804.591,E2 -7804.591} C_VEL
LIN {X 0,Y 462.147,Z 730.104,A -85,B 0,C 180,E1 -7805.519,E2 -7805.519} C_VEL
LIN {X 0,Y 461.606,Z 740.905,A -85,B 0,C 180,E1 -7806.681,E2 -7806.681} C_VEL
LIN {X 0,Y 461.139,Z 749.744,A -85,B 0,C 180,E1 -7807.864,E2 -7807.864} C_VEL
LIN {X 0,Y 460.727,Z 757.902,A -85,B 0,C 180,E1 -7809.228,E2 -7809.228} C_VEL
LIN {X 0,Y 460.363,Z 764.618,A -85,B 0,C 180,E1 -7810.631,E2 -7810.631} C_VEL
LIN {X 0,Y 460.137,Z 768.899,A -85,B 0,C 180,E1 -7811.754,E2 -7811.754} C_VEL
LIN {X 0,Y 459.957,Z 773.028,A -85,B 0,C 180,E1 -7813.124,E2 -7813.124} C_VEL
LIN {X 0,Y 459.833,Z 775.751,A -85,B 0,C 180,E1 -7814.34,E2 -7814.34} C_VEL
LIN {X 0,Y 459.674,Z 778.025,A -85,B 0,C 180,E1 -7815.841,E2 -7815.841} C_VEL
LIN {X 0,Y 459.671,Z 778.82,A -85,B 0,C 180,E1 -7816.742,E2 -7816.742} C_VEL
LIN {X 0,Y 459.694,Z 779.151,A -85,B 0,C 180,E1 -7818.536,E2 -7818.536} C_VEL
LIN {X 0,Y 459.703,Z 778.734,A -85,B 0,C 180,E1 -7819.429,E2 -7819.429} C_VEL
LIN {X 0,Y 459.754,Z 776.623,A -85,B 0,C 180,E1 -7821.207,E2 -7821.207} C_VEL
LIN {X 0,Y 459.916,Z 773.952,A -85,B 0,C 180,E1 -7822.537,E2 -7822.537} C_VEL
LIN {X 0,Y 460.047,Z 770.288,A -85,B 0,C 180,E1 -7823.861,E2 -7823.861} C_VEL
LIN {X 0,Y 460.252,Z 765.525,A -85,B 0,C 180,E1 -7825.182,E2 -7825.182} C_VEL
LIN {X 0,Y 460.526,Z 759.534,A -85,B 0,C 180,E1 -7826.5,E2 -7826.5} C_VEL
LIN {X 0,Y 460.873,Z 752.052,A -85,B 0,C 180,E1 -7827.815,E2 -7827.815} C_VEL
LIN {X 0,Y 461.435,Z 742.696,A -85,B 0,C 180,E1 -7829.127,E2 -7829.127} C_VEL
LIN {X 0,Y 461.923,Z 733.063,A -85,B 0,C 180,E1 -7830.218,E2 -7830.218} C_VEL
LIN {X 0,Y 462.363,Z 722.277,A -85,B 0,C 180,E1 -7831.198,E2 -7831.198} C_VEL
LIN {X 0,Y 462.908,Z 711.736,A -85,B 0,C 180,E1 -7831.958,E2 -7831.958} C_VEL
LIN {X 0,Y 463.319,Z 699.122,A -85,B 0,C 180,E1 -7832.663,E2 -7832.663} C_VEL
LIN {X 0,Y 463.619,Z 686.26,A -85,B 0,C 180,E1 -7833.177,E2 -7833.177} C_VEL
LIN {X 0,Y 463.848,Z 673.84,A -85,B 0,C 180,E1 -7833.502,E2 -7833.502} C_VEL
LIN {X 0,Y 464.533,Z 584.52,A -85,B 0,C 180,E1 -7834.895,E2 -7834.895} C_VEL
LIN {X 0,Y 460.679,Z 573.101,A -85,B 0,C 180,E1 -7835.224,E2 -7835.224} C_VEL
LIN {X 0,Y 460.667,Z 573.105,A -85,B 0,C 180,E1 -7837.892,E2 -7837.892} C_VEL
LIN {X 0,Y 460.632,Z 573.104,A -85,B 0,C 180,E1 -7841.44,E2 -7841.44} C_VEL
LIN {X 0,Y 460.558,Z 573.119,A -85,B 0,C 180,E1 -7844.132,E2 -7844.132} C_VEL
LIN {X 0,Y 460.567,Z 573.112,A -85,B 0,C 180,E1 -7846.853,E2 -7846.853} C_VEL
LIN {X 0,Y 460.57,Z 573.113,A -85,B 0,C 180,E1 -7849.615,E2 -7849.615} C_VEL
LIN {X 0,Y 460.511,Z 573.121,A -85,B 0,C 180,E1 -7852.428,E2 -7852.428} C_VEL
LIN {X 0,Y 460.553,Z 573.118,A -85,B 0,C 180,E1 -7855.797,E2 -7855.797} C_VEL
LIN {X 0,Y 460.573,Z 573.115,A -85,B 0,C 180,E1 -7858.822,E2 -7858.822} C_VEL
LIN {X 0,Y 464.619,Z 584.506,A -85,B 0,C 180,E1 -7859.177,E2 -7859.177} C_VEL
LIN {X 0,Y 463.685,Z 676.69,A -85,B 0,C 180,E1 -7860.67,E2 -7860.67} C_VEL
LIN {X 0,Y 463.465,Z 690.641,A -85,B 0,C 180,E1 -7861.094,E2 -7861.094} C_VEL
LIN {X 0,Y 463.186,Z 702.314,A -85,B 0,C 180,E1 -7861.617,E2 -7861.617} C_VEL
LIN {X 0,Y 462.711,Z 714.784,A -85,B 0,C 180,E1 -7862.37,E2 -7862.37} C_VEL
LIN {X 0,Y 462.203,Z 726.705,A -85,B 0,C 180,E1 -7863.305,E2 -7863.305} C_VEL
LIN {X 0,Y 461.742,Z 736.53,A -85,B 0,C 180,E1 -7864.274,E2 -7864.274} C_VEL
LIN {X 0,Y 461.251,Z 745.64,A -85,B 0,C 180,E1 -7865.379,E2 -7865.379} C_VEL
LIN {X 0,Y 460.797,Z 754.684,A -85,B 0,C 180,E1 -7866.736,E2 -7866.736} C_VEL
LIN {X 0,Y 460.467,Z 760.959,A -85,B 0,C 180,E1 -7867.902,E2 -7867.902} C_VEL
LIN {X 0,Y 460.204,Z 767.188,A -85,B 0,C 180,E1 -7869.346,E2 -7869.346} C_VEL
LIN {X 0,Y 460,Z 771.425,A -85,B 0,C 180,E1 -7870.596,E2 -7870.596} C_VEL
LIN {X 0,Y 459.798,Z 775.544,A -85,B 0,C 180,E1 -7872.262,E2 -7872.262} C_VEL
LIN {X 0,Y 459.674,Z 778.297,A -85,B 0,C 180,E1 -7874.062,E2 -7874.062} C_VEL
LIN {X 0,Y 459.623,Z 779.21,A -85,B 0,C 180,E1 -7875.301,E2 -7875.301} C_VEL
LIN {X 0,Y 459.634,Z 779.303,A -85,B 0,C 180,E1 -7876.522,E2 -7876.522} C_VEL
LIN {X 0,Y 459.676,Z 778.667,A -85,B 0,C 180,E1 -7877.723,E2 -7877.723} C_VEL
LIN {X 0,Y 459.704,Z 777.349,A -85,B 0,C 180,E1 -7878.899,E2 -7878.899} C_VEL
LIN {X 0,Y 459.894,Z 773.966,A -85,B 0,C 180,E1 -7880.64,E2 -7880.64} C_VEL
LIN {X 0,Y 460.167,Z 768.966,A -85,B 0,C 180,E1 -7882.345,E2 -7882.345} C_VEL
LIN {X 0,Y 460.402,Z 763.334,A -85,B 0,C 180,E1 -7883.764,E2 -7883.764} C_VEL
LIN {X 0,Y 460.716,Z 756.942,A -85,B 0,C 180,E1 -7885.041,E2 -7885.041} C_VEL
LIN {X 0,Y 461.098,Z 749.841,A -85,B 0,C 180,E1 -7886.198,E2 -7886.198} C_VEL
LIN {X 0,Y 461.584,Z 740.727,A -85,B 0,C 180,E1 -7887.411,E2 -7887.411} C_VEL
LIN {X 0,Y 462.118,Z 730.243,A -85,B 0,C 180,E1 -7888.522,E2 -7888.522} C_VEL
LIN {X 0,Y 462.595,Z 719.907,A -85,B 0,C 180,E1 -7889.406,E2 -7889.406} C_VEL
LIN {X 0,Y 463.027,Z 708.315,A -85,B 0,C 180,E1 -7890.192,E2 -7890.192} C_VEL
LIN {X 0,Y 463.44,Z 695.359,A -85,B 0,C 180,E1 -7890.845,E2 -7890.845} C_VEL
LIN {X 0,Y 463.681,Z 682.548,A -85,B 0,C 180,E1 -7891.302,E2 -7891.302} C_VEL
LIN {X 0,Y 463.872,Z 668.731,A -85,B 0,C 180,E1 -7891.595,E2 -7891.595} C_VEL
LIN {X 0,Y 464.657,Z 584.421,A -85,B 0,C 180,E1 -7892.954,E2 -7892.954} C_VEL
LIN {X 0,Y 460.615,Z 573.111,A -85,B 0,C 180,E1 -7893.311,E2 -7893.311} C_VEL
LIN {X 0,Y 460.538,Z 573.12,A -85,B 0,C 180,E1 -7896.623,E2 -7896.623} C_VEL
LIN {X 0,Y 460.543,Z 573.116,A -85,B 0,C 180,E1 -7899.452,E2 -7899.452} C_VEL
LIN {X 0,Y 460.55,Z 573.118,A -85,B 0,C 180,E1 -7902.23,E2 -7902.23} C_VEL
LIN {X 0,Y 460.556,Z 573.117,A -85,B 0,C 180,E1 -7904.964,E2 -7904.964} C_VEL
LIN {X 0,Y 460.648,Z 573.102,A -85,B 0,C 180,E1 -7907.667,E2 -7907.667} C_VEL
LIN {X 0,Y 460.62,Z 573.106,A -85,B 0,C 180,E1 -7911.224,E2 -7911.224} C_VEL
LIN {X 0,Y 460.707,Z 573.095,A -85,B 0,C 180,E1 -7913.87,E2 -7913.87} C_VEL
LIN {X 0,Y 460.817,Z 573.078,A -85,B 0,C 180,E1 -7917.378,E2 -7917.378} C_VEL
LIN {X 0,Y 460.843,Z 573.079,A -85,B 0,C 180,E1 -7920,E2 -7920} C_VEL
LIN {X 0,Y 460.816,Z 573.084,A -85,B 0,C 180,E1 -7922.622,E2 -7922.622} C_VEL
LIN {X 0,Y 460.708,Z 573.096,A -85,B 0,C 180,E1 -7926.13,E2 -7926.13} C_VEL
LIN {X 0,Y 460.62,Z 573.106,A -85,B 0,C 180,E1 -7928.776,E2 -7928.776} C_VEL
LIN {X 0,Y 460.625,Z 573.107,A -85,B 0,C 180,E1 -7932.457,E2 -7932.457} C_VEL
LIN {X 0,Y 460.591,Z 573.107,A -85,B 0,C 180,E1 -7935.998,E2 -7935.998} C_VEL
LIN {X 0,Y 460.562,Z 573.112,A -85,B 0,C 180,E1 -7938.902,E2 -7938.902} C_VEL
LIN {X 0,Y 460.51,Z 573.116,A -85,B 0,C 180,E1 -7941.486,E2 -7941.486} C_VEL
LIN {X 0,Y 460.536,Z 573.116,A -85,B 0,C 180,E1 -7944.333,E2 -7944.333} C_VEL
LIN {X 0,Y 460.576,Z 573.107,A -85,B 0,C 180,E1 -7947.244,E2 -7947.244} C_VEL
LIN {X 0,Y 460.52,Z 573.122,A -85,B 0,C 180,E1 -7950.239,E2 -7950.239} C_VEL
LIN {X 0,Y 460.522,Z 573.115,A -85,B 0,C 180,E1 -7953.326,E2 -7953.326} C_VEL
LIN {X 0,Y 460.474,Z 573.127,A -85,B 0,C 180,E1 -7956.53,E2 -7956.53} C_VEL
LIN {X 0,Y 460.573,Z 573.11,A -85,B 0,C 180,E1 -7959.858,E2 -7959.858} C_VEL
LIN {X 0,Y 460.538,Z 573.118,A -85,B 0,C 180,E1 -7962.905,E2 -7962.905} C_VEL
LIN {X 0,Y 460.507,Z 573.121,A -85,B 0,C 180,E1 -7965.831,E2 -7965.831} C_VEL
LIN {X 0,Y 460.535,Z 573.118,A -85,B 0,C 180,E1 -7968.99,E2 -7968.99} C_VEL
LIN {X 0,Y 460.541,Z 573.116,A -85,B 0,C 180,E1 -7971.27,E2 -7971.27} C_VEL
LIN {X 0,Y 460.509,Z 573.124,A -85,B 0,C 180,E1 -7974.555,E2 -7974.555} C_VEL
LIN {X 0,Y 460.53,Z 573.119,A -85,B 0,C 180,E1 -7977.716,E2 -7977.716} C_VEL
LIN {X 0,Y 460.552,Z 573.119,A -85,B 0,C 180,E1 -7981.27,E2 -7981.27} C_VEL
LIN {X 0,Y 460.599,Z 573.333,A -85,B 0,C 180,E1 -7981.523,E2 -7981.523} C_VEL
LIN {X 0,Y 463.226,Z 585.94,A -85,B 0,C 180,E1 -7983.714,E2 -7983.714} C_VEL
LIN {X 0,Y 463.684,Z 590.141,A -85,B 0,C 180,E1 -7984.408,E2 -7984.408} C_VEL
LIN {X 0,Y 462.732,Z 609.651,A -85,B 0,C 180,E1 -7987.45,E2 -7987.45} C_VEL
LIN {X 0,Y 461.877,Z 630.429,A -85,B 0,C 180,E1 -7990.632,E2 -7990.632} C_VEL
LIN {X 0,Y 461.343,Z 644.151,A -85,B 0,C 180,E1 -7992.694,E2 -7992.694} C_VEL
LIN {X 0,Y 464.308,Z 668.225,A -85,B 0,C 180,E1 -7993.204,E2 -7993.204} C_VEL
LIN {X 0,Y 463.53,Z 753.746,A -85,B 0,C 180,E1 -7994.585,E2 -7994.585} C_VEL
LIN {X 0,Y 463.14,Z 767.018,A -85,B 0,C 180,E1 -7994.966,E2 -7994.966} C_VEL
LIN {X 0,Y 462.681,Z 779.259,A -85,B 0,C 180,E1 -7995.486,E2 -7995.486} C_VEL
LIN {X 0,Y 462.151,Z 790.836,A -85,B 0,C 180,E1 -7996.143,E2 -7996.143} C_VEL
LIN {X 0,Y 461.621,Z 802.49,A -85,B 0,C 180,E1 -7997.002,E2 -7997.002} C_VEL
LIN {X 0,Y 461.031,Z 813.429,A -85,B 0,C 180,E1 -7998.013,E2 -7998.013} C_VEL
LIN {X 0,Y 460.649,Z 822.193,A -85,B 0,C 180,E1 -7999.006,E2 -7999.006} C_VEL
LIN {X 0,Y 460.293,Z 830.282,A -85,B 0,C 180,E1 -8000.109,E2 -8000.109} C_VEL
LIN {X 0,Y 460.035,Z 838.207,A -85,B 0,C 180,E1 -8001.434,E2 -8001.434} C_VEL
LIN {X 0,Y 459.845,Z 845.499,A -85,B 0,C 180,E1 -8002.977,E2 -8002.977} C_VEL
LIN {X 0,Y 459.756,Z 850.367,A -85,B 0,C 180,E1 -8004.298,E2 -8004.298} C_VEL
LIN {X 0,Y 459.649,Z 854.093,A -85,B 0,C 180,E1 -8005.616,E2 -8005.616} C_VEL
LIN {X 0,Y 459.698,Z 856.029,A -85,B 0,C 180,E1 -8006.494,E2 -8006.494} C_VEL
LIN {X 0,Y 459.747,Z 857.483,A -85,B 0,C 180,E1 -8007.372,E2 -8007.372} C_VEL
LIN {X 0,Y 459.57,Z 859.147,A -85,B 0,C 180,E1 -8009.124,E2 -8009.124} C_VEL
LIN {X 0,Y 459.559,Z 859.384,A -85,B 0,C 180,E1 -8010,E2 -8010} C_VEL
LIN {X 0,Y 459.637,Z 858.576,A -85,B 0,C 180,E1 -8011.752,E2 -8011.752} C_VEL
LIN {X 0,Y 459.747,Z 857.58,A -85,B 0,C 180,E1 -8012.628,E2 -8012.628} C_VEL
LIN {X 0,Y 459.694,Z 856.155,A -85,B 0,C 180,E1 -8013.506,E2 -8013.506} C_VEL
LIN {X 0,Y 459.644,Z 853.166,A -85,B 0,C 180,E1 -8014.824,E2 -8014.824} C_VEL
LIN {X 0,Y 459.709,Z 849.122,A -85,B 0,C 180,E1 -8016.143,E2 -8016.143} C_VEL
LIN {X 0,Y 459.868,Z 842.884,A -85,B 0,C 180,E1 -8017.685,E2 -8017.685} C_VEL
LIN {X 0,Y 460.096,Z 836.081,A -85,B 0,C 180,E1 -8019.008,E2 -8019.008} C_VEL
LIN {X 0,Y 460.443,Z 827.645,A -85,B 0,C 180,E1 -8020.331,E2 -8020.331} C_VEL
LIN {X 0,Y 460.904,Z 818.973,A -85,B 0,C 180,E1 -8021.433,E2 -8021.433} C_VEL
LIN {X 0,Y 461.337,Z 809.233,A -85,B 0,C 180,E1 -8022.448,E2 -8022.448} C_VEL
LIN {X 0,Y 461.771,Z 799.127,A -85,B 0,C 180,E1 -8023.308,E2 -8023.308} C_VEL
LIN {X 0,Y 462.303,Z 787.853,A -85,B 0,C 180,E1 -8024.077,E2 -8024.077} C_VEL
LIN {X 0,Y 462.893,Z 775.226,A -85,B 0,C 180,E1 -8024.732,E2 -8024.732} C_VEL
LIN {X 0,Y 463.258,Z 762.633,A -85,B 0,C 180,E1 -8025.199,E2 -8025.199} C_VEL
LIN {X 0,Y 463.631,Z 749.938,A -85,B 0,C 180,E1 -8025.496,E2 -8025.496} C_VEL
LIN {X 0,Y 464.199,Z 663.719,A -85,B 0,C 180,E1 -8026.879,E2 -8026.879} C_VEL
LIN {X 0,Y 461.826,Z 644.237,A -85,B 0,C 180,E1 -8027.291,E2 -8027.291} C_VEL
LIN {X 0,Y 462.837,Z 618.816,A -85,B 0,C 180,E1 -8030.673,E2 -8030.673} C_VEL
LIN {X 0,Y 463.97,Z 594.835,A -85,B 0,C 180,E1 -8033.903,E2 -8033.903} C_VEL
LIN {X 0,Y 464.076,Z 589.164,A -85,B 0,C 180,E1 -8034.681,E2 -8034.681} C_VEL
LIN {X 0,Y 460.668,Z 573.103,A -85,B 0,C 180,E1 -8037.114,E2 -8037.114} C_VEL
LIN {X 0,Y 460.51,Z 573.124,A -85,B 0,C 180,E1 -8040.239,E2 -8040.239} C_VEL
LIN {X 0,Y 460.528,Z 573.118,A -85,B 0,C 180,E1 -8043.324,E2 -8043.324} C_VEL
LIN {X 0,Y 460.477,Z 573.125,A -85,B 0,C 180,E1 -8046.528,E2 -8046.528} C_VEL
LIN {X 0,Y 460.571,Z 573.115,A -85,B 0,C 180,E1 -8049.857,E2 -8049.857} C_VEL
LIN {X 0,Y 460.509,Z 573.118,A -85,B 0,C 180,E1 -8052.9,E2 -8052.9} C_VEL
LIN {X 0,Y 460.519,Z 573.118,A -85,B 0,C 180,E1 -8055.828,E2 -8055.828} C_VEL
LIN {X 0,Y 460.538,Z 573.113,A -85,B 0,C 180,E1 -8058.989,E2 -8058.989} C_VEL
LIN {X 0,Y 460.542,Z 573.111,A -85,B 0,C 180,E1 -8061.268,E2 -8061.268} C_VEL
LIN {X 0,Y 460.507,Z 573.115,A -85,B 0,C 180,E1 -8064.554,E2 -8064.554} C_VEL
LIN {X 0,Y 460.525,Z 573.116,A -85,B 0,C 180,E1 -8067.715,E2 -8067.715} C_VEL
LIN {X 0,Y 460.539,Z 573.109,A -85,B 0,C 180,E1 -8070.769,E2 -8070.769} C_VEL
LIN {X 0,Y 460.56,Z 573.112,A -85,B 0,C 180,E1 -8073.734,E2 -8073.734} C_VEL
LIN {X 0,Y 460.537,Z 573.109,A -85,B 0,C 180,E1 -8076.623,E2 -8076.623} C_VEL
LIN {X 0,Y 460.543,Z 573.112,A -85,B 0,C 180,E1 -8079.452,E2 -8079.452} C_VEL
LIN {X 0,Y 460.551,Z 573.117,A -85,B 0,C 180,E1 -8082.23,E2 -8082.23} C_VEL
LIN {X 0,Y 460.555,Z 573.111,A -85,B 0,C 180,E1 -8084.964,E2 -8084.964} C_VEL
LIN {X 0,Y 460.603,Z 573.111,A -85,B 0,C 180,E1 -8088.559,E2 -8088.559} C_VEL
LIN {X 0,Y 460.685,Z 573.089,A -85,B 0,C 180,E1 -8092.108,E2 -8092.108} C_VEL
LIN {X 0,Y 460.698,Z 573.101,A -85,B 0,C 180,E1 -8094.748,E2 -8094.748} C_VEL
LIN {X 0,Y 460.817,Z 573.072,A -85,B 0,C 180,E1 -8097.378,E2 -8097.378} C_VEL
LIN {X 0,Y 460.843,Z 573.072,A -85,B 0,C 180,E1 -8100,E2 -8100} C_VEL
LIN {X 0,Y 460.816,Z 573.086,A -85,B 0,C 180,E1 -8102.622,E2 -8102.622} C_VEL
LIN {X 0,Y 460.704,Z 573.083,A -85,B 0,C 180,E1 -8106.13,E2 -8106.13} C_VEL
LIN {X 0,Y 460.62,Z 573.11,A -85,B 0,C 180,E1 -8108.776,E2 -8108.776} C_VEL
LIN {X 0,Y 460.603,Z 573.102,A -85,B 0,C 180,E1 -8112.445,E2 -8112.445} C_VEL
LIN {X 0,Y 460.591,Z 573.108,A -85,B 0,C 180,E1 -8115.998,E2 -8115.998} C_VEL
LIN {X 0,Y 460.562,Z 573.109,A -85,B 0,C 180,E1 -8118.902,E2 -8118.902} C_VEL
LIN {X 0,Y 460.507,Z 573.121,A -85,B 0,C 180,E1 -8121.486,E2 -8121.486} C_VEL
LIN {X 0,Y 460.534,Z 573.111,A -85,B 0,C 180,E1 -8124.333,E2 -8124.333} C_VEL
LIN {X 0,Y 460.577,Z 573.115,A -85,B 0,C 180,E1 -8127.244,E2 -8127.244} C_VEL
LIN {X 0,Y 460.523,Z 573.111,A -85,B 0,C 180,E1 -8130.239,E2 -8130.239} C_VEL
LIN {X 0,Y 460.522,Z 573.118,A -85,B 0,C 180,E1 -8133.326,E2 -8133.326} C_VEL
LIN {X 0,Y 460.473,Z 573.124,A -85,B 0,C 180,E1 -8136.53,E2 -8136.53} C_VEL
LIN {X 0,Y 460.561,Z 573.11,A -85,B 0,C 180,E1 -8139.859,E2 -8139.859} C_VEL
LIN {X 0,Y 460.512,Z 573.106,A -85,B 0,C 180,E1 -8142.902,E2 -8142.902} C_VEL
LIN {X 0,Y 460.505,Z 573.119,A -85,B 0,C 180,E1 -8145.831,E2 -8145.831} C_VEL
LIN {X 0,Y 460.527,Z 573.114,A -85,B 0,C 180,E1 -8148.99,E2 -8148.99} C_VEL
LIN {X 0,Y 460.524,Z 573.118,A -85,B 0,C 180,E1 -8151.268,E2 -8151.268} C_VEL
LIN {X 0,Y 460.512,Z 573.118,A -85,B 0,C 180,E1 -8154.556,E2 -8154.556} C_VEL
LIN {X 0,Y 460.53,Z 573.121,A -85,B 0,C 180,E1 -8157.716,E2 -8157.716} C_VEL
LIN {X 0,Y 460.552,Z 573.116,A -85,B 0,C 180,E1 -8160.755,E2 -8160.755} C_VEL
LIN {X 0,Y 464.744,Z 584.599,A -85,B 0,C 180,E1 -8161.13,E2 -8161.13} C_VEL
LIN {X 0,Y 463.934,Z 675.903,A -85,B 0,C 180,E1 -8162.574,E2 -8162.574} C_VEL
LIN {X 0,Y 463.696,Z 688.875,A -85,B 0,C 180,E1 -8162.94,E2 -8162.94} C_VEL
LIN {X 0,Y 463.419,Z 701.401,A -85,B 0,C 180,E1 -8163.479,E2 -8163.479} C_VEL
LIN {X 0,Y 463.193,Z 707.557,A -85,B 0,C 180,E1 -8163.815,E2 -8163.815} C_VEL
LIN {X 0,Y 462.412,Z 712.94,A -85,B 0,C 180,E1 -8164.125,E2 -8164.125} C_VEL
LIN {X 0,Y 459.204,Z 721.443,A -85,B 0,C 180,E1 -8164.633,E2 -8164.633} C_VEL
LIN {X 0,Y 455.969,Z 729.51,A -85,B 0,C 180,E1 -8165.22,E2 -8165.22} C_VEL
LIN {X 0,Y 455.115,Z 734.136,A -85,B 0,C 180,E1 -8165.654,E2 -8165.654} C_VEL
LIN {X 0,Y 454.599,Z 743.821,A -85,B 0,C 180,E1 -8166.783,E2 -8166.783} C_VEL
LIN {X 0,Y 454.102,Z 752.042,A -85,B 0,C 180,E1 -8167.957,E2 -8167.957} C_VEL
LIN {X 0,Y 453.628,Z 760.016,A -85,B 0,C 180,E1 -8169.363,E2 -8169.363} C_VEL
LIN {X 0,Y 453.358,Z 765.351,A -85,B 0,C 180,E1 -8170.532,E2 -8170.532} C_VEL
LIN {X 0,Y 453.065,Z 770.459,A -85,B 0,C 180,E1 -8171.927,E2 -8171.927} C_VEL
LIN {X 0,Y 452.905,Z 774.332,A -85,B 0,C 180,E1 -8173.317,E2 -8173.317} C_VEL
LIN {X 0,Y 452.733,Z 777.12,A -85,B 0,C 180,E1 -8174.699,E2 -8174.699} C_VEL
LIN {X 0,Y 452.623,Z 778.414,A -85,B 0,C 180,E1 -8175.615,E2 -8175.615} C_VEL
LIN {X 0,Y 452.607,Z 779.302,A -85,B 0,C 180,E1 -8176.531,E2 -8176.531} C_VEL
LIN {X 0,Y 452.637,Z 779.839,A -85,B 0,C 180,E1 -8178.012,E2 -8178.012} C_VEL
LIN {X 0,Y 452.629,Z 779.435,A -85,B 0,C 180,E1 -8179.262,E2 -8179.262} C_VEL
LIN {X 0,Y 452.614,Z 778.693,A -85,B 0,C 180,E1 -8180.166,E2 -8180.166} C_VEL
LIN {X 0,Y 452.684,Z 777.5,A -85,B 0,C 180,E1 -8181.069,E2 -8181.069} C_VEL
LIN {X 0,Y 452.825,Z 774.956,A -85,B 0,C 180,E1 -8182.419,E2 -8182.419} C_VEL
LIN {X 0,Y 452.99,Z 771.419,A -85,B 0,C 180,E1 -8183.765,E2 -8183.765} C_VEL
LIN {X 0,Y 453.194,Z 766.796,A -85,B 0,C 180,E1 -8185.107,E2 -8185.107} C_VEL
LIN {X 0,Y 453.535,Z 759.877,A -85,B 0,C 180,E1 -8186.669,E2 -8186.669} C_VEL
LIN {X 0,Y 453.93,Z 752.307,A -85,B 0,C 180,E1 -8188.004,E2 -8188.004} C_VEL
LIN {X 0,Y 454.513,Z 742.88,A -85,B 0,C 180,E1 -8189.336,E2 -8189.336} C_VEL
LIN {X 0,Y 454.991,Z 733.127,A -85,B 0,C 180,E1 -8190.443,E2 -8190.443} C_VEL
LIN {X 0,Y 455.507,Z 722.203,A -85,B 0,C 180,E1 -8191.437,E2 -8191.437} C_VEL
LIN {X 0,Y 456.066,Z 711.506,A -85,B 0,C 180,E1 -8192.208,E2 -8192.208} C_VEL
LIN {X 0,Y 456.451,Z 699.718,A -85,B 0,C 180,E1 -8192.868,E2 -8192.868} C_VEL
LIN {X 0,Y 456.767,Z 686.049,A -85,B 0,C 180,E1 -8193.418,E2 -8193.418} C_VEL
LIN {X 0,Y 456.991,Z 672.978,A -85,B 0,C 180,E1 -8193.747,E2 -8193.747} C_VEL
LIN {X 0,Y 457.69,Z 585.959,A -85,B 0,C 180,E1 -8195.121,E2 -8195.121} C_VEL
LIN {X 0,Y 453.647,Z 573.978,A -85,B 0,C 180,E1 -8195.473,E2 -8195.473} C_VEL
LIN {X 0,Y 453.609,Z 573.985,A -85,B 0,C 180,E1 -8198.015,E2 -8198.015} C_VEL
LIN {X 0,Y 453.542,Z 573.987,A -85,B 0,C 180,E1 -8200.716,E2 -8200.716} C_VEL
LIN {X 0,Y 453.536,Z 573.988,A -85,B 0,C 180,E1 -8203.44,E2 -8203.44} C_VEL
LIN {X 0,Y 453.547,Z 573.992,A -85,B 0,C 180,E1 -8206.195,E2 -8206.195} C_VEL
LIN {X 0,Y 453.522,Z 573.989,A -85,B 0,C 180,E1 -8209.04,E2 -8209.04} C_VEL
LIN {X 0,Y 453.477,Z 573.998,A -85,B 0,C 180,E1 -8211.836,E2 -8211.836} C_VEL
LIN {X 0,Y 453.5,Z 573.992,A -85,B 0,C 180,E1 -8214.735,E2 -8214.735} C_VEL
LIN {X 0,Y 453.533,Z 573.992,A -85,B 0,C 180,E1 -8218.249,E2 -8218.249} C_VEL
LIN {X 0,Y 453.527,Z 573.994,A -85,B 0,C 180,E1 -8218.566,E2 -8218.566} C_VEL
LIN {X 0,Y 457.731,Z 585.723,A -85,B 0,C 180,E1 -8218.934,E2 -8218.934} C_VEL
LIN {X 0,Y 456.87,Z 676.029,A -85,B 0,C 180,E1 -8220.416,E2 -8220.416} C_VEL
LIN {X 0,Y 456.665,Z 689.404,A -85,B 0,C 180,E1 -8220.809,E2 -8220.809} C_VEL
LIN {X 0,Y 456.368,Z 701.961,A -85,B 0,C 180,E1 -8221.359,E2 -8221.359} C_VEL
LIN {X 0,Y 455.939,Z 713.328,A -85,B 0,C 180,E1 -8222.028,E2 -8222.028} C_VEL
LIN {X 0,Y 455.466,Z 723.82,A -85,B 0,C 180,E1 -8222.817,E2 -8222.817} C_VEL
LIN {X 0,Y 454.966,Z 734.151,A -85,B 0,C 180,E1 -8223.786,E2 -8223.786} C_VEL
LIN {X 0,Y 454.416,Z 744.154,A -85,B 0,C 180,E1 -8224.945,E2 -8224.945} C_VEL
LIN {X 0,Y 453.964,Z 752.862,A -85,B 0,C 180,E1 -8226.201,E2 -8226.201} C_VEL
LIN {X 0,Y 453.514,Z 760.019,A -85,B 0,C 180,E1 -8227.474,E2 -8227.474} C_VEL
LIN {X 0,Y 453.282,Z 765.785,A -85,B 0,C 180,E1 -8228.741,E2 -8228.741} C_VEL
LIN {X 0,Y 453.008,Z 770.409,A -85,B 0,C 180,E1 -8230,E2 -8230} C_VEL
LIN {X 0,Y 452.875,Z 774.008,A -85,B 0,C 180,E1 -8231.249,E2 -8231.249} C_VEL
LIN {X 0,Y 452.715,Z 776.689,A -85,B 0,C 180,E1 -8232.476,E2 -8232.476} C_VEL
LIN {X 0,Y 452.679,Z 777.787,A -85,B 0,C 180,E1 -8233.139,E2 -8233.139} C_VEL
LIN {X 0,Y 452.595,Z 779.257,A -85,B 0,C 180,E1 -8234.414,E2 -8234.414} C_VEL
LIN {X 0,Y 452.569,Z 779.914,A -85,B 0,C 180,E1 -8235.668,E2 -8235.668} C_VEL
LIN {X 0,Y 452.563,Z 779.818,A -85,B 0,C 180,E1 -8236.898,E2 -8236.898} C_VEL
LIN {X 0,Y 452.63,Z 778.911,A -85,B 0,C 180,E1 -8238.183,E2 -8238.183} C_VEL
LIN {X 0,Y 452.709,Z 777.056,A -85,B 0,C 180,E1 -8239.523,E2 -8239.523} C_VEL
LIN {X 0,Y 452.887,Z 774.186,A -85,B 0,C 180,E1 -8240.886,E2 -8240.886} C_VEL
LIN {X 0,Y 453.118,Z 770.157,A -85,B 0,C 180,E1 -8242.28,E2 -8242.28} C_VEL
LIN {X 0,Y 453.393,Z 763.844,A -85,B 0,C 180,E1 -8243.911,E2 -8243.911} C_VEL
LIN {X 0,Y 453.739,Z 757.608,A -85,B 0,C 180,E1 -8245.175,E2 -8245.175} C_VEL
LIN {X 0,Y 454.193,Z 749.942,A -85,B 0,C 180,E1 -8246.437,E2 -8246.437} C_VEL
LIN {X 0,Y 454.661,Z 741.114,A -85,B 0,C 180,E1 -8247.618,E2 -8247.618} C_VEL
LIN {X 0,Y 455.239,Z 730.762,A -85,B 0,C 180,E1 -8248.728,E2 -8248.728} C_VEL
LIN {X 0,Y 455.803,Z 719.371,A -85,B 0,C 180,E1 -8249.705,E2 -8249.705} C_VEL
LIN {X 0,Y 456.214,Z 708.01,A -85,B 0,C 180,E1 -8250.464,E2 -8250.464} C_VEL
LIN {X 0,Y 456.657,Z 695.01,A -85,B 0,C 180,E1 -8251.115,E2 -8251.115} C_VEL
LIN {X 0,Y 456.876,Z 682.748,A -85,B 0,C 180,E1 -8251.55,E2 -8251.55} C_VEL
LIN {X 0,Y 457.089,Z 667.621,A -85,B 0,C 180,E1 -8251.862,E2 -8251.862} C_VEL
LIN {X 0,Y 457.825,Z 585.668,A -85,B 0,C 180,E1 -8253.211,E2 -8253.211} C_VEL
LIN {X 0,Y 453.547,Z 573.999,A -85,B 0,C 180,E1 -8253.593,E2 -8253.593} C_VEL
LIN {X 0,Y 453.495,Z 573.998,A -85,B 0,C 180,E1 -8256.238,E2 -8256.238} C_VEL
LIN {X 0,Y 453.474,Z 573.999,A -85,B 0,C 180,E1 -8259.117,E2 -8259.117} C_VEL
LIN {X 0,Y 453.503,Z 573.994,A -85,B 0,C 180,E1 -8261.944,E2 -8261.944} C_VEL
LIN {X 0,Y 453.53,Z 573.994,A -85,B 0,C 180,E1 -8264.726,E2 -8264.726} C_VEL
LIN {X 0,Y 453.593,Z 573.981,A -85,B 0,C 180,E1 -8267.472,E2 -8267.472} C_VEL
LIN {X 0,Y 453.584,Z 573.984,A -85,B 0,C 180,E1 -8271.086,E2 -8271.086} C_VEL
LIN {X 0,Y 453.673,Z 573.971,A -85,B 0,C 180,E1 -8273.775,E2 -8273.775} C_VEL
LIN {X 0,Y 453.757,Z 573.958,A -85,B 0,C 180,E1 -8277.337,E2 -8277.337} C_VEL
LIN {X 0,Y 453.814,Z 573.955,A -85,B 0,C 180,E1 -8280,E2 -8280} C_VEL
LIN {X 0,Y 453.757,Z 573.963,A -85,B 0,C 180,E1 -8282.663,E2 -8282.663} C_VEL
LIN {X 0,Y 453.674,Z 573.974,A -85,B 0,C 180,E1 -8286.225,E2 -8286.225} C_VEL
LIN {X 0,Y 453.584,Z 573.981,A -85,B 0,C 180,E1 -8288.914,E2 -8288.914} C_VEL
LIN {X 0,Y 453.592,Z 573.981,A -85,B 0,C 180,E1 -8292.551,E2 -8292.551} C_VEL
LIN {X 0,Y 453.535,Z 573.988,A -85,B 0,C 180,E1 -8296.196,E2 -8296.196} C_VEL
LIN {X 0,Y 453.511,Z 573.989,A -85,B 0,C 180,E1 -8299.041,E2 -8299.041} C_VEL
LIN {X 0,Y 453.47,Z 573.994,A -85,B 0,C 180,E1 -8301.837,E2 -8301.837} C_VEL
LIN {X 0,Y 453.507,Z 573.996,A -85,B 0,C 180,E1 -8304.735,E2 -8304.735} C_VEL
LIN {X 0,Y 453.531,Z 573.986,A -85,B 0,C 180,E1 -8307.962,E2 -8307.962} C_VEL
LIN {X 0,Y 453.476,Z 573.997,A -85,B 0,C 180,E1 -8310.76,E2 -8310.76} C_VEL
LIN {X 0,Y 453.471,Z 573.994,A -85,B 0,C 180,E1 -8313.913,E2 -8313.913} C_VEL
LIN {X 0,Y 453.466,Z 573.997,A -85,B 0,C 180,E1 -8317.189,E2 -8317.189} C_VEL
LIN {X 0,Y 453.528,Z 573.987,A -85,B 0,C 180,E1 -8319.446,E2 -8319.446} C_VEL
LIN {X 0,Y 453.487,Z 573.995,A -85,B 0,C 180,E1 -8322.992,E2 -8322.992} C_VEL
LIN {X 0,Y 453.462,Z 573.998,A -85,B 0,C 180,E1 -8325.78,E2 -8325.78} C_VEL
LIN {X 0,Y 453.513,Z 573.99,A -85,B 0,C 180,E1 -8329.407,E2 -8329.407} C_VEL
LIN {X 0,Y 453.474,Z 574.001,A -85,B 0,C 180,E1 -8332.224,E2 -8332.224} C_VEL
LIN {X 0,Y 453.486,Z 573.995,A -85,B 0,C 180,E1 -8335.223,E2 -8335.223} C_VEL
LIN {X 0,Y 453.465,Z 574.002,A -85,B 0,C 180,E1 -8338.476,E2 -8338.476} C_VEL
LIN {X 0,Y 453.544,Z 574.149,A -85,B 0,C 180,E1 -8341.26,E2 -8341.26} C_VEL
LIN {X 0,Y 456.205,Z 586.529,A -85,B 0,C 180,E1 -8343.465,E2 -8343.465} C_VEL
LIN {X 0,Y 456.762,Z 591.088,A -85,B 0,C 180,E1 -8344.236,E2 -8344.236} C_VEL
LIN {X 0,Y 455.778,Z 610.602,A -85,B 0,C 180,E1 -8347.326,E2 -8347.326} C_VEL
LIN {X 0,Y 454.87,Z 630.77,A -85,B 0,C 180,E1 -8350.474,E2 -8350.474} C_VEL
LIN {X 0,Y 454.365,Z 643.272,A -85,B 0,C 180,E1 -8352.402,E2 -8352.402} C_VEL
LIN {X 0,Y 457.522,Z 667.785,A -85,B 0,C 180,E1 -8352.945,E2 -8352.945} C_VEL
LIN {X 0,Y 456.692,Z 753.079,A -85,B 0,C 180,E1 -8354.349,E2 -8354.349} C_VEL
LIN {X 0,Y 456.237,Z 766.32,A -85,B 0,C 180,E1 -8354.733,E2 -8354.733} C_VEL
LIN {X 0,Y 455.762,Z 778.549,A -85,B 0,C 180,E1 -8355.26,E2 -8355.26} C_VEL
LIN {X 0,Y 455.221,Z 790.125,A -85,B 0,C 180,E1 -8355.927,E2 -8355.927} C_VEL
LIN {X 0,Y 454.667,Z 801.2,A -85,B 0,C 180,E1 -8356.749,E2 -8356.749} C_VEL
LIN {X 0,Y 454.169,Z 811.651,A -85,B 0,C 180,E1 -8357.715,E2 -8357.715} C_VEL
LIN {X 0,Y 453.635,Z 821.511,A -85,B 0,C 180,E1 -8358.834,E2 -8358.834} C_VEL
LIN {X 0,Y 453.234,Z 829.609,A -85,B 0,C 180,E1 -8359.954,E2 -8359.954} C_VEL
LIN {X 0,Y 452.964,Z 837.547,A -85,B 0,C 180,E1 -8361.299,E2 -8361.299} C_VEL
LIN {X 0,Y 452.756,Z 844.852,A -85,B 0,C 180,E1 -8362.867,E2 -8362.867} C_VEL
LIN {X 0,Y 452.672,Z 849.729,A -85,B 0,C 180,E1 -8364.208,E2 -8364.208} C_VEL
LIN {X 0,Y 452.561,Z 853.462,A -85,B 0,C 180,E1 -8365.547,E2 -8365.547} C_VEL
LIN {X 0,Y 452.63,Z 855.404,A -85,B 0,C 180,E1 -8366.439,E2 -8366.439} C_VEL
LIN {X 0,Y 452.674,Z 856.861,A -85,B 0,C 180,E1 -8367.33,E2 -8367.33} C_VEL
LIN {X 0,Y 452.579,Z 857.893,A -85,B 0,C 180,E1 -8368.22,E2 -8368.22} C_VEL
LIN {X 0,Y 452.504,Z 858.53,A -85,B 0,C 180,E1 -8369.11,E2 -8369.11} C_VEL
LIN {X 0,Y 452.491,Z 858.768,A -85,B 0,C 180,E1 -8370,E2 -8370} C_VEL
LIN {X 0,Y 452.579,Z 857.961,A -85,B 0,C 180,E1 -8371.78,E2 -8371.78} C_VEL
LIN {X 0,Y 452.673,Z 856.964,A -85,B 0,C 180,E1 -8372.67,E2 -8372.67} C_VEL
LIN {X 0,Y 452.627,Z 855.537,A -85,B 0,C 180,E1 -8373.561,E2 -8373.561} C_VEL
LIN {X 0,Y 452.577,Z 852.545,A -85,B 0,C 180,E1 -8374.899,E2 -8374.899} C_VEL
LIN {X 0,Y 452.691,Z 847.604,A -85,B 0,C 180,E1 -8376.486,E2 -8376.486} C_VEL
LIN {X 0,Y 452.844,Z 841.221,A -85,B 0,C 180,E1 -8378.029,E2 -8378.029} C_VEL
LIN {X 0,Y 453.078,Z 834.175,A -85,B 0,C 180,E1 -8379.373,E2 -8379.373} C_VEL
LIN {X 0,Y 453.495,Z 825.348,A -85,B 0,C 180,E1 -8380.717,E2 -8380.717} C_VEL
LIN {X 0,Y 453.962,Z 815.326,A -85,B 0,C 180,E1 -8381.95,E2 -8381.95} C_VEL
LIN {X 0,Y 454.473,Z 805.214,A -85,B 0,C 180,E1 -8382.953,E2 -8382.953} C_VEL
LIN {X 0,Y 455.097,Z 793.893,A -85,B 0,C 180,E1 -8383.849,E2 -8383.849} C_VEL
LIN {X 0,Y 455.614,Z 783.268,A -85,B 0,C 180,E1 -8384.516,E2 -8384.516} C_VEL
LIN {X 0,Y 456.062,Z 770.505,A -85,B 0,C 180,E1 -8385.13,E2 -8385.13} C_VEL
LIN {X 0,Y 456.561,Z 757.879,A -85,B 0,C 180,E1 -8385.541,E2 -8385.541} C_VEL
LIN {X 0,Y 456.867,Z 740.23,A -85,B 0,C 180,E1 -8385.874,E2 -8385.874} C_VEL
LIN {X 0,Y 457.423,Z 664.987,A -85,B 0,C 180,E1 -8387.099,E2 -8387.099} C_VEL
LIN {X 0,Y 454.833,Z 643.614,A -85,B 0,C 180,E1 -8387.565,E2 -8387.565} C_VEL
LIN {X 0,Y 455.861,Z 619.921,A -85,B 0,C 180,E1 -8390.768,E2 -8390.768} C_VEL
LIN {X 0,Y 457.077,Z 595.975,A -85,B 0,C 180,E1 -8394.045,E2 -8394.045} C_VEL
LIN {X 0,Y 457.241,Z 591.189,A -85,B 0,C 180,E1 -8394.709,E2 -8394.709} C_VEL
LIN {X 0,Y 454.197,Z 576.738,A -85,B 0,C 180,E1 -8396.91,E2 -8396.91} C_VEL
LIN {X 0,Y 453.602,Z 573.983,A -85,B 0,C 180,E1 -8397.353,E2 -8397.353} C_VEL
LIN {X 0,Y 453.475,Z 573.997,A -85,B 0,C 180,E1 -8400.759,E2 -8400.759} C_VEL
LIN {X 0,Y 453.477,Z 574.001,A -85,B 0,C 180,E1 -8403.912,E2 -8403.912} C_VEL
LIN {X 0,Y 453.469,Z 573.996,A -85,B 0,C 180,E1 -8407.187,E2 -8407.187} C_VEL
LIN {X 0,Y 453.525,Z 573.988,A -85,B 0,C 180,E1 -8409.445,E2 -8409.445} C_VEL
LIN {X 0,Y 453.475,Z 573.996,A -85,B 0,C 180,E1 -8411.934,E2 -8411.934} C_VEL
LIN {X 0,Y 453.489,Z 573.991,A -85,B 0,C 180,E1 -8415.469,E2 -8415.469} C_VEL
LIN {X 0,Y 453.492,Z 573.999,A -85,B 0,C 180,E1 -8418.21,E2 -8418.21} C_VEL
LIN {X 0,Y 453.527,Z 573.986,A -85,B 0,C 180,E1 -8420.787,E2 -8420.787} C_VEL
LIN {X 0,Y 453.451,Z 574.001,A -85,B 0,C 180,E1 -8423.917,E2 -8423.917} C_VEL
LIN {X 0,Y 453.476,Z 573.993,A -85,B 0,C 180,E1 -8427.151,E2 -8427.151} C_VEL
LIN {X 0,Y 453.507,Z 573.989,A -85,B 0,C 180,E1 -8430.27,E2 -8430.27} C_VEL
LIN {X 0,Y 453.506,Z 573.99,A -85,B 0,C 180,E1 -8433.294,E2 -8433.294} C_VEL
LIN {X 0,Y 453.495,Z 573.992,A -85,B 0,C 180,E1 -8436.238,E2 -8436.238} C_VEL
LIN {X 0,Y 453.474,Z 573.994,A -85,B 0,C 180,E1 -8439.117,E2 -8439.117} C_VEL
LIN {X 0,Y 453.503,Z 573.992,A -85,B 0,C 180,E1 -8441.944,E2 -8441.944} C_VEL
LIN {X 0,Y 453.53,Z 573.985,A -85,B 0,C 180,E1 -8444.726,E2 -8444.726} C_VEL
LIN {X 0,Y 453.552,Z 573.99,A -85,B 0,C 180,E1 -8448.379,E2 -8448.379} C_VEL
LIN {X 0,Y 453.642,Z 573.965,A -85,B 0,C 180,E1 -8451.985,E2 -8451.985} C_VEL
LIN {X 0,Y 453.671,Z 573.977,A -85,B 0,C 180,E1 -8454.667,E2 -8454.667} C_VEL
LIN {X 0,Y 453.757,Z 573.952,A -85,B 0,C 180,E1 -8457.337,E2 -8457.337} C_VEL
LIN {X 0,Y 453.814,Z 573.947,A -85,B 0,C 180,E1 -8460,E2 -8460} C_VEL
LIN {X 0,Y 453.757,Z 573.966,A -85,B 0,C 180,E1 -8462.663,E2 -8462.663} C_VEL
LIN {X 0,Y 453.671,Z 573.96,A -85,B 0,C 180,E1 -8466.225,E2 -8466.225} C_VEL
LIN {X 0,Y 453.583,Z 573.988,A -85,B 0,C 180,E1 -8468.914,E2 -8468.914} C_VEL
LIN {X 0,Y 453.554,Z 573.98,A -85,B 0,C 180,E1 -8472.529,E2 -8472.529} C_VEL
LIN {X 0,Y 453.535,Z 573.987,A -85,B 0,C 180,E1 -8476.196,E2 -8476.196} C_VEL
LIN {X 0,Y 453.511,Z 573.987,A -85,B 0,C 180,E1 -8479.041,E2 -8479.041} C_VEL
LIN {X 0,Y 453.467,Z 573.995,A -85,B 0,C 180,E1 -8481.837,E2 -8481.837} C_VEL
LIN {X 0,Y 453.506,Z 573.988,A -85,B 0,C 180,E1 -8484.735,E2 -8484.735} C_VEL
LIN {X 0,Y 453.531,Z 573.987,A -85,B 0,C 180,E1 -8487.962,E2 -8487.962} C_VEL
LIN {X 0,Y 453.478,Z 573.992,A -85,B 0,C 180,E1 -8490.76,E2 -8490.76} C_VEL
LIN {X 0,Y 453.471,Z 573.991,A -85,B 0,C 180,E1 -8493.913,E2 -8493.913} C_VEL
LIN {X 0,Y 453.465,Z 574.001,A -85,B 0,C 180,E1 -8497.189,E2 -8497.189} C_VEL
LIN {X 0,Y 453.517,Z 573.992,A -85,B 0,C 180,E1 -8499.447,E2 -8499.447} C_VEL
LIN {X 0,Y 453.473,Z 573.98,A -85,B 0,C 180,E1 -8501.936,E2 -8501.936} C_VEL
LIN {X 0,Y 453.482,Z 573.998,A -85,B 0,C 180,E1 -8505.472,E2 -8505.472} C_VEL
LIN {X 0,Y 453.475,Z 573.989,A -85,B 0,C 180,E1 -8508.21,E2 -8508.21} C_VEL
LIN {X 0,Y 453.507,Z 573.993,A -85,B 0,C 180,E1 -8510.792,E2 -8510.792} C_VEL
LIN {X 0,Y 453.455,Z 574,A -85,B 0,C 180,E1 -8513.918,E2 -8513.918} C_VEL
LIN {X 0,Y 453.481,Z 573.999,A -85,B 0,C 180,E1 -8517.152,E2 -8517.152} C_VEL
LIN {X 0,Y 453.502,Z 574.077,A -85,B 0,C 180,E1 -8520.472,E2 -8520.472} C_VEL
LIN {X 0,Y 458.019,Z 586.35,A -85,B 0,C 180,E1 -8520.874,E2 -8520.874} C_VEL
LIN {X 0,Y 457.105,Z 677.707,A -85,B 0,C 180,E1 -8522.347,E2 -8522.347} C_VEL
LIN {X 0,Y 456.905,Z 689.933,A -85,B 0,C 180,E1 -8522.709,E2 -8522.709} C_VEL
LIN {X 0,Y 456.573,Z 702.799,A -85,B 0,C 180,E1 -8523.281,E2 -8523.281} C_VEL
LIN {X 0,Y 456.165,Z 714.036,A -85,B 0,C 180,E1 -8523.955,E2 -8523.955} C_VEL
LIN {X 0,Y 455.641,Z 724.872,A -85,B 0,C 180,E1 -8524.78,E2 -8524.78} C_VEL
LIN {X 0,Y 455.115,Z 734.136,A -85,B 0,C 180,E1 -8525.654,E2 -8525.654} C_VEL
LIN {X 0,Y 454.298,Z 738.685,A -85,B 0,C 180,E1 -8526.118,E2 -8526.118} C_VEL
LIN {X 0,Y 451.115,Z 745.796,A -85,B 0,C 180,E1 -8526.896,E2 -8526.896} C_VEL
LIN {X 0,Y 447.872,Z 752.339,A -85,B 0,C 180,E1 -8527.754,E2 -8527.754} C_VEL
LIN {X 0,Y 446.974,Z 755.977,A -85,B 0,C 180,E1 -8528.339,E2 -8528.339} C_VEL
LIN {X 0,Y 446.515,Z 763.144,A -85,B 0,C 180,E1 -8529.741,E2 -8529.741} C_VEL
LIN {X 0,Y 446.155,Z 769.261,A -85,B 0,C 180,E1 -8531.274,E2 -8531.274} C_VEL
LIN {X 0,Y 445.921,Z 773.294,A -85,B 0,C 180,E1 -8532.576,E2 -8532.576} C_VEL
LIN {X 0,Y 445.751,Z 776.796,A -85,B 0,C 180,E1 -8534.106,E2 -8534.106} C_VEL
LIN {X 0,Y 445.579,Z 778.809,A -85,B 0,C 180,E1 -8535.383,E2 -8535.383} C_VEL
LIN {X 0,Y 445.549,Z 779.757,A -85,B 0,C 180,E1 -8536.314,E2 -8536.314} C_VEL
LIN {X 0,Y 445.578,Z 780.435,A -85,B 0,C 180,E1 -8537.936,E2 -8537.936} C_VEL
LIN {X 0,Y 445.567,Z 780.128,A -85,B 0,C 180,E1 -8539.09,E2 -8539.09} C_VEL
LIN {X 0,Y 445.537,Z 779.458,A -85,B 0,C 180,E1 -8540.008,E2 -8540.008} C_VEL
LIN {X 0,Y 445.607,Z 778.372,A -85,B 0,C 180,E1 -8540.926,E2 -8540.926} C_VEL
LIN {X 0,Y 445.699,Z 776.842,A -85,B 0,C 180,E1 -8541.841,E2 -8541.841} C_VEL
LIN {X 0,Y 445.907,Z 773.806,A -85,B 0,C 180,E1 -8543.195,E2 -8543.195} C_VEL
LIN {X 0,Y 446.058,Z 769.656,A -85,B 0,C 180,E1 -8544.576,E2 -8544.576} C_VEL
LIN {X 0,Y 446.371,Z 763.419,A -85,B 0,C 180,E1 -8546.163,E2 -8546.163} C_VEL
LIN {X 0,Y 446.768,Z 756.566,A -85,B 0,C 180,E1 -8547.521,E2 -8547.521} C_VEL
LIN {X 0,Y 447.216,Z 748.055,A -85,B 0,C 180,E1 -8548.874,E2 -8548.874} C_VEL
LIN {X 0,Y 447.783,Z 739.327,A -85,B 0,C 180,E1 -8550,E2 -8550} C_VEL
LIN {X 0,Y 448.24,Z 729.765,A -85,B 0,C 180,E1 -8551.011,E2 -8551.011} C_VEL
LIN {X 0,Y 448.826,Z 719.195,A -85,B 0,C 180,E1 -8551.907,E2 -8551.907} C_VEL
LIN {X 0,Y 449.377,Z 707.498,A -85,B 0,C 180,E1 -8552.689,E2 -8552.689} C_VEL
LIN {X 0,Y 449.729,Z 695.397,A -85,B 0,C 180,E1 -8553.303,E2 -8553.303} C_VEL
LIN {X 0,Y 450.045,Z 681.82,A -85,B 0,C 180,E1 -8553.777,E2 -8553.777} C_VEL
LIN {X 0,Y 450.193,Z 668.33,A -85,B 0,C 180,E1 -8554.056,E2 -8554.056} C_VEL
LIN {X 0,Y 450.946,Z 587.904,A -85,B 0,C 180,E1 -8555.337,E2 -8555.337} C_VEL
LIN {X 0,Y 446.613,Z 574.855,A -85,B 0,C 180,E1 -8555.715,E2 -8555.715} C_VEL
LIN {X 0,Y 446.576,Z 574.861,A -85,B 0,C 180,E1 -8558.142,E2 -8558.142} C_VEL
LIN {X 0,Y 446.541,Z 574.863,A -85,B 0,C 180,E1 -8561.806,E2 -8561.806} C_VEL
LIN {X 0,Y 446.51,Z 574.864,A -85,B 0,C 180,E1 -8565.52,E2 -8565.52} C_VEL
LIN {X 0,Y 446.459,Z 574.873,A -85,B 0,C 180,E1 -8568.35,E2 -8568.35} C_VEL
LIN {X 0,Y 446.449,Z 574.873,A -85,B 0,C 180,E1 -8571.754,E2 -8571.754} C_VEL
LIN {X 0,Y 446.444,Z 574.871,A -85,B 0,C 180,E1 -8575.152,E2 -8575.152} C_VEL
LIN {X 0,Y 446.513,Z 574.994,A -85,B 0,C 180,E1 -8578.304,E2 -8578.304} C_VEL
LIN {X 0,Y 450.979,Z 587.375,A -85,B 0,C 180,E1 -8578.696,E2 -8578.696} C_VEL
LIN {X 0,Y 449.985,Z 677.981,A -85,B 0,C 180,E1 -8580.221,E2 -8580.221} C_VEL
LIN {X 0,Y 449.77,Z 691.393,A -85,B 0,C 180,E1 -8580.64,E2 -8580.64} C_VEL
LIN {X 0,Y 449.458,Z 703.507,A -85,B 0,C 180,E1 -8581.195,E2 -8581.195} C_VEL
LIN {X 0,Y 449.013,Z 714.795,A -85,B 0,C 180,E1 -8581.887,E2 -8581.887} C_VEL
LIN {X 0,Y 448.505,Z 725.531,A -85,B 0,C 180,E1 -8582.725,E2 -8582.725} C_VEL
LIN {X 0,Y 447.968,Z 736.039,A -85,B 0,C 180,E1 -8583.747,E2 -8583.747} C_VEL
LIN {X 0,Y 447.37,Z 746.109,A -85,B 0,C 180,E1 -8584.967,E2 -8584.967} C_VEL
LIN {X 0,Y 446.856,Z 755.347,A -85,B 0,C 180,E1 -8586.375,E2 -8586.375} C_VEL
LIN {X 0,Y 446.457,Z 761.78,A -85,B 0,C 180,E1 -8587.588,E2 -8587.588} C_VEL
LIN {X 0,Y 446.175,Z 768.039,A -85,B 0,C 180,E1 -8589.054,E2 -8589.054} C_VEL
LIN {X 0,Y 445.919,Z 772.08,A -85,B 0,C 180,E1 -8590.254,E2 -8590.254} C_VEL
LIN {X 0,Y 445.77,Z 775.284,A -85,B 0,C 180,E1 -8591.464,E2 -8591.464} C_VEL
LIN {X 0,Y 445.633,Z 777.746,A -85,B 0,C 180,E1 -8592.698,E2 -8592.698} C_VEL
LIN {X 0,Y 445.542,Z 779.467,A -85,B 0,C 180,E1 -8593.951,E2 -8593.951} C_VEL
LIN {X 0,Y 445.489,Z 780.408,A -85,B 0,C 180,E1 -8595.227,E2 -8595.227} C_VEL
LIN {X 0,Y 445.477,Z 780.545,A -85,B 0,C 180,E1 -8596.527,E2 -8596.527} C_VEL
LIN {X 0,Y 445.545,Z 779.857,A -85,B 0,C 180,E1 -8597.847,E2 -8597.847} C_VEL
LIN {X 0,Y 445.687,Z 777.441,A -85,B 0,C 180,E1 -8599.72,E2 -8599.72} C_VEL
LIN {X 0,Y 445.939,Z 773.453,A -85,B 0,C 180,E1 -8601.486,E2 -8601.486} C_VEL
LIN {X 0,Y 446.259,Z 767.74,A -85,B 0,C 180,E1 -8603.241,E2 -8603.241} C_VEL
LIN {X 0,Y 446.579,Z 761.501,A -85,B 0,C 180,E1 -8604.686,E2 -8604.686} C_VEL
LIN {X 0,Y 446.973,Z 754.396,A -85,B 0,C 180,E1 -8606,E2 -8606} C_VEL
LIN {X 0,Y 447.614,Z 745.379,A -85,B 0,C 180,E1 -8607.335,E2 -8607.335} C_VEL
LIN {X 0,Y 448.096,Z 736.193,A -85,B 0,C 180,E1 -8608.435,E2 -8608.435} C_VEL
LIN {X 0,Y 448.691,Z 725.382,A -85,B 0,C 180,E1 -8609.481,E2 -8609.481} C_VEL
LIN {X 0,Y 449.183,Z 714.128,A -85,B 0,C 180,E1 -8610.343,E2 -8610.343} C_VEL
LIN {X 0,Y 449.695,Z 701.755,A -85,B 0,C 180,E1 -8611.065,E2 -8611.065} C_VEL
LIN {X 0,Y 449.931,Z 689.076,A -85,B 0,C 180,E1 -8611.612,E2 -8611.612} C_VEL
LIN {X 0,Y 450.19,Z 675.63,A -85,B 0,C 180,E1 -8611.979,E2 -8611.979} C_VEL
LIN {X 0,Y 451.203,Z 587.555,A -85,B 0,C 180,E1 -8613.459,E2 -8613.459} C_VEL
LIN {X 0,Y 446.514,Z 574.867,A -85,B 0,C 180,E1 -8613.895,E2 -8613.895} C_VEL
LIN {X 0,Y 446.421,Z 574.879,A -85,B 0,C 180,E1 -8616.823,E2 -8616.823} C_VEL
LIN {X 0,Y 446.436,Z 574.874,A -85,B 0,C 180,E1 -8619.737,E2 -8619.737} C_VEL
LIN {X 0,Y 446.455,Z 574.877,A -85,B 0,C 180,E1 -8622.597,E2 -8622.597} C_VEL
LIN {X 0,Y 446.463,Z 574.87,A -85,B 0,C 180,E1 -8625.412,E2 -8625.412} C_VEL
LIN {X 0,Y 446.537,Z 574.864,A -85,B 0,C 180,E1 -8628.194,E2 -8628.194} C_VEL
LIN {X 0,Y 446.591,Z 574.854,A -85,B 0,C 180,E1 -8631.858,E2 -8631.858} C_VEL
LIN {X 0,Y 446.643,Z 574.85,A -85,B 0,C 180,E1 -8634.583,E2 -8634.583} C_VEL
LIN {X 0,Y 446.701,Z 574.837,A -85,B 0,C 180,E1 -8637.295,E2 -8637.295} C_VEL
LIN {X 0,Y 446.784,Z 574.83,A -85,B 0,C 180,E1 -8640,E2 -8640} C_VEL
LIN {X 0,Y 446.701,Z 574.841,A -85,B 0,C 180,E1 -8642.705,E2 -8642.705} C_VEL
LIN {X 0,Y 446.642,Z 574.849,A -85,B 0,C 180,E1 -8646.324,E2 -8646.324} C_VEL
LIN {X 0,Y 446.53,Z 574.858,A -85,B 0,C 180,E1 -8649.056,E2 -8649.056} C_VEL
LIN {X 0,Y 446.524,Z 574.859,A -85,B 0,C 180,E1 -8652.73,E2 -8652.73} C_VEL
LIN {X 0,Y 446.481,Z 574.866,A -85,B 0,C 180,E1 -8656.459,E2 -8656.459} C_VEL
LIN {X 0,Y 446.461,Z 574.865,A -85,B 0,C 180,E1 -8659.304,E2 -8659.304} C_VEL
LIN {X 0,Y 446.413,Z 574.876,A -85,B 0,C 180,E1 -8662.2,E2 -8662.2} C_VEL
LIN {X 0,Y 446.451,Z 574.871,A -85,B 0,C 180,E1 -8665.153,E2 -8665.153} C_VEL
LIN {X 0,Y 446.477,Z 574.867,A -85,B 0,C 180,E1 -8668.179,E2 -8668.179} C_VEL
LIN {X 0,Y 446.413,Z 574.874,A -85,B 0,C 180,E1 -8671.301,E2 -8671.301} C_VEL
LIN {X 0,Y 446.424,Z 574.878,A -85,B 0,C 180,E1 -8674.524,E2 -8674.524} C_VEL
LIN {X 0,Y 446.433,Z 574.875,A -85,B 0,C 180,E1 -8678.084,E2 -8678.084} C_VEL
LIN {X 0,Y 446.442,Z 574.872,A -85,B 0,C 180,E1 -8680.921,E2 -8680.921} C_VEL
LIN {X 0,Y 446.441,Z 574.872,A -85,B 0,C 180,E1 -8683.841,E2 -8683.841} C_VEL
LIN {X 0,Y 446.395,Z 574.883,A -85,B 0,C 180,E1 -8686.404,E2 -8686.404} C_VEL
LIN {X 0,Y 446.465,Z 574.869,A -85,B 0,C 180,E1 -8689.806,E2 -8689.806} C_VEL
LIN {X 0,Y 446.43,Z 574.877,A -85,B 0,C 180,E1 -8692.124,E2 -8692.124} C_VEL
LIN {X 0,Y 446.427,Z 574.875,A -85,B 0,C 180,E1 -8695.478,E2 -8695.478} C_VEL
LIN {X 0,Y 446.415,Z 574.879,A -85,B 0,C 180,E1 -8698.7,E2 -8698.7} C_VEL
LIN {X 0,Y 446.474,Z 574.876,A -85,B 0,C 180,E1 -8700.972,E2 -8700.972} C_VEL
LIN {X 0,Y 449.479,Z 589.193,A -85,B 0,C 180,E1 -8703.562,E2 -8703.562} C_VEL
LIN {X 0,Y 449.793,Z 593.562,A -85,B 0,C 180,E1 -8704.305,E2 -8704.305} C_VEL
LIN {X 0,Y 448.778,Z 612.27,A -85,B 0,C 180,E1 -8707.317,E2 -8707.317} C_VEL
LIN {X 0,Y 447.813,Z 632.944,A -85,B 0,C 180,E1 -8710.596,E2 -8710.596} C_VEL
LIN {X 0,Y 447.374,Z 642.547,A -85,B 0,C 180,E1 -8712.103,E2 -8712.103} C_VEL
LIN {X 0,Y 450.711,Z 669.264,A -85,B 0,C 180,E1 -8712.709,E2 -8712.709} C_VEL
LIN {X 0,Y 449.833,Z 752.492,A -85,B 0,C 180,E1 -8714.104,E2 -8714.104} C_VEL
LIN {X 0,Y 449.408,Z 765.703,A -85,B 0,C 180,E1 -8714.496,E2 -8714.496} C_VEL
LIN {X 0,Y 448.872,Z 777.915,A -85,B 0,C 180,E1 -8715.029,E2 -8715.029} C_VEL
LIN {X 0,Y 448.3,Z 789.484,A -85,B 0,C 180,E1 -8715.705,E2 -8715.705} C_VEL
LIN {X 0,Y 447.686,Z 801.114,A -85,B 0,C 180,E1 -8716.588,E2 -8716.588} C_VEL
LIN {X 0,Y 447.124,Z 812.086,A -85,B 0,C 180,E1 -8717.634,E2 -8717.634} C_VEL
LIN {X 0,Y 446.632,Z 820.853,A -85,B 0,C 180,E1 -8718.657,E2 -8718.657} C_VEL
LIN {X 0,Y 446.201,Z 828.949,A -85,B 0,C 180,E1 -8719.794,E2 -8719.794} C_VEL
LIN {X 0,Y 445.877,Z 836.886,A -85,B 0,C 180,E1 -8721.16,E2 -8721.16} C_VEL
LIN {X 0,Y 445.681,Z 844.205,A -85,B 0,C 180,E1 -8722.753,E2 -8722.753} C_VEL
LIN {X 0,Y 445.572,Z 849.09,A -85,B 0,C 180,E1 -8724.116,E2 -8724.116} C_VEL
LIN {X 0,Y 445.478,Z 852.833,A -85,B 0,C 180,E1 -8725.476,E2 -8725.476} C_VEL
LIN {X 0,Y 445.564,Z 854.779,A -85,B 0,C 180,E1 -8726.383,E2 -8726.383} C_VEL
LIN {X 0,Y 445.589,Z 856.237,A -85,B 0,C 180,E1 -8727.288,E2 -8727.288} C_VEL
LIN {X 0,Y 445.522,Z 857.276,A -85,B 0,C 180,E1 -8728.192,E2 -8728.192} C_VEL
LIN {X 0,Y 445.442,Z 857.915,A -85,B 0,C 180,E1 -8729.096,E2 -8729.096} C_VEL
LIN {X 0,Y 445.425,Z 858.153,A -85,B 0,C 180,E1 -8730,E2 -8730} C_VEL
LIN {X 0,Y 445.522,Z 857.348,A -85,B 0,C 180,E1 -8731.808,E2 -8731.808} C_VEL
LIN {X 0,Y 445.589,Z 856.347,A -85,B 0,C 180,E1 -8732.712,E2 -8732.712} C_VEL
LIN {X 0,Y 445.56,Z 854.919,A -85,B 0,C 180,E1 -8733.617,E2 -8733.617} C_VEL
LIN {X 0,Y 445.514,Z 851.923,A -85,B 0,C 180,E1 -8734.977,E2 -8734.977} C_VEL
LIN {X 0,Y 445.605,Z 847.398,A -85,B 0,C 180,E1 -8736.471,E2 -8736.471} C_VEL
LIN {X 0,Y 445.721,Z 841.606,A -85,B 0,C 180,E1 -8737.93,E2 -8737.93} C_VEL
LIN {X 0,Y 445.976,Z 834.785,A -85,B 0,C 180,E1 -8739.295,E2 -8739.295} C_VEL
LIN {X 0,Y 446.365,Z 826.323,A -85,B 0,C 180,E1 -8740.661,E2 -8740.661} C_VEL
LIN {X 0,Y 446.859,Z 817.615,A -85,B 0,C 180,E1 -8741.797,E2 -8741.797} C_VEL
LIN {X 0,Y 447.371,Z 807.932,A -85,B 0,C 180,E1 -8742.834,E2 -8742.834} C_VEL
LIN {X 0,Y 447.978,Z 796.265,A -85,B 0,C 180,E1 -8743.842,E2 -8743.842} C_VEL
LIN {X 0,Y 448.612,Z 784.494,A -85,B 0,C 180,E1 -8744.632,E2 -8744.632} C_VEL
LIN {X 0,Y 449.107,Z 772.277,A -85,B 0,C 180,E1 -8745.253,E2 -8745.253} C_VEL
LIN {X 0,Y 449.644,Z 759.003,A -85,B 0,C 180,E1 -8745.728,E2 -8745.728} C_VEL
LIN {X 0,Y 449.926,Z 746.012,A -85,B 0,C 180,E1 -8746.009,E2 -8746.009} C_VEL
LIN {X 0,Y 450.651,Z 665.958,A -85,B 0,C 180,E1 -8747.332,E2 -8747.332} C_VEL
LIN {X 0,Y 447.88,Z 643.137,A -85,B 0,C 180,E1 -8747.827,E2 -8747.827} C_VEL
LIN {X 0,Y 448.897,Z 621.03,A -85,B 0,C 180,E1 -8750.865,E2 -8750.865} C_VEL
LIN {X 0,Y 450.159,Z 597.074,A -85,B 0,C 180,E1 -8754.193,E2 -8754.193} C_VEL
LIN {X 0,Y 450.243,Z 591.905,A -85,B 0,C 180,E1 -8754.926,E2 -8754.926} C_VEL
LIN {X 0,Y 446.817,Z 576.083,A -85,B 0,C 180,E1 -8757.391,E2 -8757.391} C_VEL
LIN {X 0,Y 446.52,Z 574.866,A -85,B 0,C 180,E1 -8757.601,E2 -8757.601} C_VEL
LIN {X 0,Y 446.426,Z 574.878,A -85,B 0,C 180,E1 -8760.249,E2 -8760.249} C_VEL
LIN {X 0,Y 446.443,Z 574.873,A -85,B 0,C 180,E1 -8763.453,E2 -8763.453} C_VEL
LIN {X 0,Y 446.407,Z 574.876,A -85,B 0,C 180,E1 -8766.744,E2 -8766.744} C_VEL
LIN {X 0,Y 446.486,Z 574.866,A -85,B 0,C 180,E1 -8769.529,E2 -8769.529} C_VEL
LIN {X 0,Y 446.426,Z 574.874,A -85,B 0,C 180,E1 -8772.604,E2 -8772.604} C_VEL
LIN {X 0,Y 446.452,Z 574.867,A -85,B 0,C 180,E1 -8775.102,E2 -8775.102} C_VEL
LIN {X 0,Y 446.439,Z 574.872,A -85,B 0,C 180,E1 -8778.61,E2 -8778.61} C_VEL
LIN {X 0,Y 446.47,Z 574.864,A -85,B 0,C 180,E1 -8780.976,E2 -8780.976} C_VEL
LIN {X 0,Y 446.415,Z 574.872,A -85,B 0,C 180,E1 -8784.373,E2 -8784.373} C_VEL
LIN {X 0,Y 446.422,Z 574.873,A -85,B 0,C 180,E1 -8787.638,E2 -8787.638} C_VEL
LIN {X 0,Y 446.462,Z 574.862,A -85,B 0,C 180,E1 -8790.791,E2 -8790.791} C_VEL
LIN {X 0,Y 446.47,Z 574.868,A -85,B 0,C 180,E1 -8793.848,E2 -8793.848} C_VEL
LIN {X 0,Y 446.42,Z 574.865,A -85,B 0,C 180,E1 -8796.823,E2 -8796.823} C_VEL
LIN {X 0,Y 446.435,Z 574.87,A -85,B 0,C 180,E1 -8799.737,E2 -8799.737} C_VEL
LIN {X 0,Y 446.454,Z 574.867,A -85,B 0,C 180,E1 -8802.597,E2 -8802.597} C_VEL
LIN {X 0,Y 446.462,Z 574.863,A -85,B 0,C 180,E1 -8805.412,E2 -8805.412} C_VEL
LIN {X 0,Y 446.509,Z 574.865,A -85,B 0,C 180,E1 -8808.193,E2 -8808.193} C_VEL
LIN {X 0,Y 446.591,Z 574.842,A -85,B 0,C 180,E1 -8811.858,E2 -8811.858} C_VEL
LIN {X 0,Y 446.644,Z 574.851,A -85,B 0,C 180,E1 -8814.583,E2 -8814.583} C_VEL
LIN {X 0,Y 446.701,Z 574.831,A -85,B 0,C 180,E1 -8817.295,E2 -8817.295} C_VEL
LIN {X 0,Y 446.785,Z 574.823,A -85,B 0,C 180,E1 -8820,E2 -8820} C_VEL
LIN {X 0,Y 446.701,Z 574.845,A -85,B 0,C 180,E1 -8822.705,E2 -8822.705} C_VEL
LIN {X 0,Y 446.64,Z 574.836,A -85,B 0,C 180,E1 -8826.324,E2 -8826.324} C_VEL
LIN {X 0,Y 446.529,Z 574.864,A -85,B 0,C 180,E1 -8829.056,E2 -8829.056} C_VEL
LIN {X 0,Y 446.512,Z 574.857,A -85,B 0,C 180,E1 -8832.73,E2 -8832.73} C_VEL
LIN {X 0,Y 446.487,Z 574.866,A -85,B 0,C 180,E1 -8836.228,E2 -8836.228} C_VEL
LIN {X 0,Y 446.46,Z 574.866,A -85,B 0,C 180,E1 -8839.304,E2 -8839.304} C_VEL
LIN {X 0,Y 446.409,Z 574.875,A -85,B 0,C 180,E1 -8842.2,E2 -8842.2} C_VEL
LIN {X 0,Y 446.45,Z 574.869,A -85,B 0,C 180,E1 -8845.153,E2 -8845.153} C_VEL
LIN {X 0,Y 446.477,Z 574.866,A -85,B 0,C 180,E1 -8848.179,E2 -8848.179} C_VEL
LIN {X 0,Y 446.427,Z 574.878,A -85,B 0,C 180,E1 -8851.3,E2 -8851.3} C_VEL
LIN {X 0,Y 446.424,Z 574.869,A -85,B 0,C 180,E1 -8854.524,E2 -8854.524} C_VEL
LIN {X 0,Y 446.426,Z 574.872,A -85,B 0,C 180,E1 -8858.083,E2 -8858.083} C_VEL
LIN {X 0,Y 446.437,Z 574.868,A -85,B 0,C 180,E1 -8860.921,E2 -8860.921} C_VEL
LIN {X 0,Y 446.418,Z 574.874,A -85,B 0,C 180,E1 -8863.844,E2 -8863.844} C_VEL
LIN {X 0,Y 446.394,Z 574.875,A -85,B 0,C 180,E1 -8866.404,E2 -8866.404} C_VEL
LIN {X 0,Y 446.423,Z 574.872,A -85,B 0,C 180,E1 -8869.083,E2 -8869.083} C_VEL
LIN {X 0,Y 446.425,Z 574.868,A -85,B 0,C 180,E1 -8872.124,E2 -8872.124} C_VEL
LIN {X 0,Y 446.429,Z 574.878,A -85,B 0,C 180,E1 -8875.478,E2 -8875.478} C_VEL
LIN {X 0,Y 446.415,Z 574.875,A -85,B 0,C 180,E1 -8878.7,E2 -8878.7} C_VEL
LIN {X 0,Y 446.424,Z 574.876,A -85,B 0,C 180,E1 -8880.149,E2 -8880.149} C_VEL
LIN {X 0,Y 448.817,Z 581.267,A -85,B 0,C 180,E1 -8880.378,E2 -8880.378} C_VEL
LIN {X 0,Y 451.332,Z 588.015,A -85,B 0,C 180,E1 -8880.606,E2 -8880.606} C_VEL
LIN {X 0,Y 450.348,Z 678.39,A -85,B 0,C 180,E1 -8882.085,E2 -8882.085} C_VEL
LIN {X 0,Y 450.147,Z 690.963,A -85,B 0,C 180,E1 -8882.467,E2 -8882.467} C_VEL
LIN {X 0,Y 449.769,Z 703.829,A -85,B 0,C 180,E1 -8883.055,E2 -8883.055} C_VEL
LIN {X 0,Y 449.305,Z 715.541,A -85,B 0,C 180,E1 -8883.777,E2 -8883.777} C_VEL
